  MoveL 5894 to (-63.02, -0.01, -9) mm, rotated rx -180 ry 0 rz 90 deg; joints [73.202, -18.477, 88.716, 0, 19.76, 73.202]
  MoveL 5895 to (-27.01, 8.34, -9) mm, rotated rx -180 ry 0 rz 90 deg; joints [73.832, -17.933, 86.424, 0, 21.509, 73.832]
  MoveL 5896 to (-22.05, 9.5, -9) mm, rotated rx 180 ry 0 rz 90 deg; joints [73.917, -17.854, 86.103, 0, 21.751, 73.917]
  MoveC 5897 to (-21.12, 9.91, -9) mm, rotated rx 180 ry 0 rz 90 deg; joints [73.939, -17.84, 86.046, 0, 21.794, 73.939] to (-20.37, 10.6, -9) mm, rotated rx 180 ry 0 rz 90 deg; joints [73.969, -17.83, 86.008, 0, 21.822, 73.969]
  MoveC 5898 to (-19.58, 12.14, -9) mm, rotated rx -180 ry 0 rz 90 deg; joints [74.027, -17.824, 85.984, 0, 21.841, 74.027] to (-19.7, 13.87, -9) mm, rotated rx 180 ry 0 rz 90 deg; joints [74.082, -17.835, 86.026, 0, 21.809, 74.082]
  MoveL 5899 to (-19.98, 14.69, -9) mm, rotated rx 180 ry 0 rz 90 deg; joints [74.107, -17.844, 86.062, 0, 21.782, 74.107]
  MoveL 5900 to (-26.01, 31.57, -9) mm, rotated rx 180 ry 0 rz 90 deg; joints [74.608, -18.027, 86.81, 0, 21.218, 74.608]
  MoveC 5901 to (-26.34, 32.29, -9) mm, rotated rx 180 ry 0 rz 90 deg; joints [74.628, -18.036, 86.846, 0, 21.19, 74.628] to (-26.8, 32.94, -9) mm, rotated rx -180 ry 0 rz 90 deg; joints [74.646, -18.047, 86.89, 0, 21.156, 74.646]
  MoveL 5902 to (-27.74, 33.64, -9) mm, rotated rx 180 ry 0 rz 90 deg; joints [74.66, -18.066, 86.969, 0, 21.097, 74.66]
  MoveL 5903 to (-62.07, 55.73, -9) mm, rotated rx -180 ry 0 rz 90 deg; joints [75.091, -18.703, 89.719, 0, 18.983, 75.091]
  MoveL 5904 to (-69.19, 60.28, -9) mm, rotated rx 180 ry 0 rz 90 deg; joints [75.181, -18.825, 90.278, 0, 18.547, 75.181]
  MoveC 5905 to (-69.62, 60.48, -9) mm, rotated rx -180 ry 0 rz 90 deg; joints [75.184, -18.832, 90.311, 0, 18.521, 75.184] to (-70.09, 60.56, -9) mm, rotated rx -180 ry 0 rz 90 deg; joints [75.183, -18.84, 90.344, 0, 18.496, 75.183]
  MoveC 5906 to (-72.08, 60.11, -9) mm, rotated rx 180 ry 0 rz 90 deg; joints [75.149, -18.867, 90.469, 0, 18.397, 75.149] to (-73.6, 58.75, -9) mm, rotated rx 180 ry 0 rz 90 deg; joints [75.089, -18.883, 90.547, 0, 18.337, 75.089]
  MoveC 5907 to (-73.89, 58.14, -9) mm, rotated rx 180 ry 0 rz 90 deg; joints [75.065, -18.885, 90.555, 0, 18.33, 75.065] to (-73.99, 57.48, -9) mm, rotated rx -180 ry 0 rz 90 deg; joints [75.042, -18.884, 90.55, 0, 18.334, 75.042]
  MoveL 5908 to (-73.99, 29.63, -9) mm, rotated rx 180 ry 0 rz 90 deg; joints [74.092, -18.773, 90.036, 0, 18.736, 74.092]
  MoveL 5909 to (-66.44, 29.63, -9) mm, rotated rx -180 ry 0 rz 90 deg; joints [74.165, -18.661, 89.531, 0, 19.13, 74.165]
  MoveL 5910 to (-66.44, 29.63, -6) mm, rotated rx -180 ry 0 rz 90 deg; joints [74.165, -18.818, 89.632, 0, 19.185, 74.165]
  Establecer velocidad (1000.0 mm/s)
  MoveL 5911 to (-66.44, 29.63, 10) mm, rotated rx 180 ry 0 rz 90 deg; joints [74.165, -19.655, 90.167, 0, 19.487, 74.165]
  Establecer velocidad (66.7 mm/s)
  MoveL 5912 to (-39.77, -31.53, 10) mm, rotated rx -180 ry 0 rz 90 deg; joints [72.398, -18.924, 87.105, 0, 21.819, 72.398]
  MoveL 5913 to (-39.77, -31.53, -5.75) mm, rotated rx -180 ry 0 rz 90 deg; joints [72.398, -18.112, 86.579, 0, 21.532, 72.398]
  MoveL 5914 to (-39.9, -30.02, -6.16) mm, rotated rx 180 ry 0 rz 90 deg; joints [72.446, -18.101, 86.607, 0, 21.494, 72.446]
  MoveL 5915 to (-40.39, -28.58, -6.56) mm, rotated rx -180 ry 0 rz 90 deg; joints [72.488, -18.096, 86.659, 0, 21.437, 72.488]
  MoveL 5916 to (-41.19, -27.29, -6.97) mm, rotated rx -180 ry 0 rz 90 deg; joints [72.522, -18.095, 86.728, 0, 21.368, 72.522]
  MoveL 5917 to (-42.25, -26.2, -7.38) mm, rotated rx -180 ry 0 rz 90 deg; joints [72.547, -18.098, 86.81, 0, 21.287, 72.547]
  MoveL 5918 to (-43.53, -25.38, -7.78) mm, rotated rx 180 ry 0 rz 90 deg; joints [72.561, -18.102, 86.902, 0, 21.201, 72.561]
  MoveL 5919 to (-44.95, -24.86, -8.19) mm, rotated rx 180 ry 0 rz 90 deg; joints [72.563, -18.108, 86.997, 0, 21.111, 72.563]
  MoveL 5920 to (-46.46, -24.67, -8.59) mm, rotated rx 180 ry 0 rz 90 deg; joints [72.554, -18.113, 87.09, 0, 21.022, 72.554]
  MoveL 5921 to (-47.97, -24.84, -9) mm, rotated rx 180 ry 0 rz 90 deg; joints [72.533, -18.116, 87.176, 0, 20.94, 72.533]
  MoveL 5922 to (-71.48, -29.8, -9) mm, rotated rx -180 ry 0 rz 90 deg; joints [72.121, -18.464, 88.66, 0, 19.804, 72.121]
  MoveC 5923 to (-73.12, -30.73, -9) mm, rotated rx -180 ry 0 rz 90 deg; joints [72.073, -18.485, 88.75, 0, 19.735, 72.073] to (-73.94, -32.43, -9) mm, rotated rx 180 ry 0 rz 90 deg; joints [72.008, -18.489, 88.768, 0, 19.721, 72.008]
  MoveC 5924 to (-73.98, -32.78, -9) mm, rotated rx 180 ry 0 rz 90 deg; joints [71.996, -18.487, 88.763, 0, 19.725, 71.996] to (-73.99, -33.14, -9) mm, rotated rx 180 ry 0 rz 90 deg; joints [71.983, -18.486, 88.756, 0, 19.73, 71.983]
  MoveL 5925 to (-73.99, -70.1, -9) mm, rotated rx 180 ry 0 rz 90 deg; joints [70.765, -18.292, 87.921, 0, 20.371, 70.765]
  MoveC 5926 to (-73.78, -71.26, -9) mm, rotated rx -180 ry 0 rz 90 deg; joints [70.729, -18.283, 87.88, 0, 20.403, 70.729] to (-73.19, -72.29, -9) mm, rotated rx -180 ry 0 rz 90 deg; joints [70.703, -18.268, 87.816, 0, 20.452, 70.703]
  MoveC 5927 to (-72.08, -73.13, -9) mm, rotated rx 180 ry 0 rz 90 deg; joints [70.688, -18.246, 87.722, 0, 20.524, 70.688] to (-70.73, -73.41, -9) mm, rotated rx -180 ry 0 rz 90 deg; joints [70.694, -18.223, 87.624, 0, 20.598, 70.694]
  MoveL 5928 to (-36.48, -73.09, -9) mm, rotated rx 180 ry 0 rz 90 deg; joints [71.089, -17.652, 85.298, 0, 22.355, 71.089]
  MoveL 5929 to (-35.72, -73.07, -9) mm, rotated rx 180 ry 0 rz 90 deg; joints [71.098, -17.639, 85.245, 0, 22.394, 71.098]
  MoveC 5930 to (-33.81, -72.36, -9) mm, rotated rx 180 ry 0 rz 90 deg; joints [71.141, -17.61, 85.13, 0, 22.48, 71.141] to (-32.71, -70.66, -9) mm, rotated rx 180 ry 0 rz 90 deg; joints [71.208, -17.601, 85.094, 0, 22.507, 71.208]
  MoveL 5931 to (-20.54, -23.88, -9) mm, rotated rx 180 ry 0 rz 90 deg; joints [72.843, -17.654, 85.303, 0, 22.351, 72.843]
  MoveC 5932 to (-20.49, -23.55, -9) mm, rotated rx 180 ry 0 rz 90 deg; joints [72.854, -17.655, 85.307, 0, 22.348, 72.854] to (-20.52, -23.22, -9) mm, rotated rx 180 ry 0 rz 90 deg; joints [72.865, -17.657, 85.316, 0, 22.341, 72.865]
  MoveC 5933 to (-21.45, -21.25, -9) mm, rotated rx 180 ry 0 rz 90 deg; joints [72.919, -17.684, 85.423, 0, 22.261, 72.919] to (-23.23, -19.99, -9) mm, rotated rx -180 ry 0 rz 90 deg; joints [72.942, -17.722, 85.574, 0, 22.148, 72.942]
  MoveC 5934 to (-23.83, -19.86, -9) mm, rotated rx 180 ry 0 rz 90 deg; joints [72.941, -17.733, 85.619, 0, 22.114, 72.941] to (-24.45, -19.9, -9) mm, rotated rx 180 ry 0 rz 90 deg; joints [72.933, -17.744, 85.661, 0, 22.083, 72.933]
  MoveL 5935 to (-33.64, -21.82, -9) mm, rotated rx 180 ry 0 rz 90 deg; joints [72.778, -17.892, 86.257, 0, 21.635, 72.778]
  MoveL 5936 to (-47.97, -24.84, -9) mm, rotated rx 180 ry 0 rz 90 deg; joints [72.533, -18.116, 87.176, 0, 20.94, 72.533]
  MoveL 5937 to (-46.41, -32.23, -9) mm, rotated rx 180 ry 0 rz 90 deg; joints [72.307, -18.051, 86.909, 0, 21.142, 72.307]
  MoveL 5938 to (-46.41, -32.23, -6) mm, rotated rx -180 ry 0 rz 90 deg; joints [72.307, -18.206, 87.011, 0, 21.195, 72.307]
  Establecer velocidad (1000.0 mm/s)
  MoveL 5939 to (-46.41, -32.23, 10) mm, rotated rx -180 ry 0 rz 90 deg; joints [72.307, -19.033, 87.545, 0, 21.488, 72.307]
  Establecer velocidad (66.7 mm/s)
  MoveL 5940 to (15.82, -64.4, 10) mm, rotated rx -180 ry 0 rz 90 deg; joints [71.919, -17.693, 82.448, 0, 25.246, 71.919]
  MoveL 5941 to (15.82, -64.4, -5.75) mm, rotated rx 180 ry 0 rz 90 deg; joints [71.919, -16.896, 81.92, 0, 24.977, 71.919]
  MoveL 5942 to (15.68, -65.91, -6.16) mm, rotated rx 180 ry 0 rz 90 deg; joints [71.87, -16.869, 81.881, 0, 24.988, 71.87]
  MoveL 5943 to (15.9, -67.41, -6.56) mm, rotated rx 180 ry 0 rz 90 deg; joints [71.826, -16.834, 81.815, 0, 25.019, 71.826]
  MoveL 5944 to (16.45, -68.83, -6.97) mm, rotated rx 180 ry 0 rz 90 deg; joints [71.787, -16.793, 81.728, 0, 25.065, 71.787]
  MoveL 5945 to (17.29, -70.09, -7.38) mm, rotated rx 180 ry 0 rz 90 deg; joints [71.756, -16.747, 81.623, 0, 25.124, 71.756]
  MoveL 5946 to (18.4, -71.13, -7.78) mm, rotated rx -180 ry 0 rz 90 deg; joints [71.735, -16.698, 81.504, 0, 25.194, 71.735]
  MoveL 5947 to (19.71, -71.9, -8.19) mm, rotated rx -180 ry 0 rz 90 deg; joints [71.724, -16.646, 81.377, 0, 25.269, 71.724]
  MoveL 5948 to (21.16, -72.36, -8.59) mm, rotated rx 180 ry 0 rz 90 deg; joints [71.725, -16.593, 81.247, 0, 25.346, 71.725]
  MoveL 5949 to (22.67, -72.47, -9) mm, rotated rx -180 ry 0 rz 90 deg; joints [71.737, -16.541, 81.121, 0, 25.42, 71.737]
  MoveC 5950 to (33.77, -72.15, -9) mm, rotated rx -180 ry 0 rz 90 deg; joints [71.861, -16.316, 80.318, 0, 25.998, 71.861] to (44.87, -71.79, -9) mm, rotated rx 180 ry 0 rz 90 deg; joints [71.984, -16.085, 79.509, 0, 26.576, 71.984]
  MoveC 5951 to (46.9, -69.65, -9) mm, rotated rx -180 ry 0 rz 90 deg; joints [72.07, -16.056, 79.41, 0, 26.647, 72.07] to (47.66, -66.81, -9) mm, rotated rx 180 ry 0 rz 90 deg; joints [72.165, -16.06, 79.421, 0, 26.639, 72.165]
  MoveL 5952 to (47.63, -65.95, -9) mm, rotated rx -180 ry 0 rz 90 deg; joints [72.192, -16.066, 79.444, 0, 26.622, 72.192]
  MoveC 5953 to (47.48, -65.22, -9) mm, rotated rx -180 ry 0 rz 90 deg; joints [72.213, -16.074, 79.473, 0, 26.602, 72.213] to (47.1, -64.57, -9) mm, rotated rx 180 ry 0 rz 90 deg; joints [72.229, -16.087, 79.516, 0, 26.571, 72.229]
  MoveL 5954 to (45.03, -62.07, -9) mm, rotated rx -180 ry 0 rz 90 deg; joints [72.286, -16.148, 79.729, 0, 26.419, 72.286]
  MoveL 5955 to (29.13, -43.12, -9) mm, rotated rx -180 ry 0 rz 90 deg; joints [72.72, -16.601, 81.336, 0, 25.265, 72.72]
  MoveL 5956 to (25.02, -38.27, -9) mm, rotated rx -180 ry 0 rz 90 deg; joints [72.833, -16.714, 81.744, 0, 24.969, 72.833]
  MoveC 5957 to (24.6, -37.8, -9) mm, rotated rx -180 ry 0 rz 90 deg; joints [72.844, -16.725, 81.785, 0, 24.94, 72.844] to (24.17, -37.36, -9) mm, rotated rx -180 ry 0 rz 90 deg; joints [72.853, -16.736, 81.826, 0, 24.91, 72.853]
  MoveL 5958 to (12.79, -28.13, -9) mm, rotated rx 180 ry 0 rz 90 deg; joints [73.035, -17.014, 82.851, 0, 24.163, 73.035]
  MoveC 5959 to (10.35, -27.65, -9) mm, rotated rx 180 ry 0 rz 90 deg; joints [73.027, -17.064, 83.037, 0, 24.027, 73.027] to (8.05, -28.61, -9) mm, rotated rx -180 ry 0 rz 90 deg; joints [72.974, -17.102, 83.18, 0, 23.922, 72.974]
  MoveC 5960 to (7.53, -29.2, -9) mm, rotated rx -180 ry 0 rz 90 deg; joints [72.95, -17.109, 83.205, 0, 23.904, 72.95] to (7.21, -29.92, -9) mm, rotated rx 180 ry 0 rz 90 deg; joints [72.924, -17.111, 83.212, 0, 23.899, 72.924]
  MoveL 5961 to (-2.19, -64.91, -9) mm, rotated rx 180 ry 0 rz 90 deg; joints [71.717, -17.078, 83.087, 0, 23.99, 71.717]
  MoveL 5962 to (-3.2, -68.7, -9) mm, rotated rx -180 ry 0 rz 90 deg; joints [71.586, -17.073, 83.069, 0, 24.004, 71.586]
  MoveL 5963 to (-3.29, -69.18, -9) mm, rotated rx -180 ry 0 rz 90 deg; joints [71.57, -17.072, 83.064, 0, 24.007, 71.57]
  MoveC 5964 to (-2.2, -71.85, -9) mm, rotated rx 180 ry 0 rz 90 deg; joints [71.497, -17.034, 82.923, 0, 24.11, 71.497] to (0.47, -72.94, -9) mm, rotated rx 180 ry 0 rz 90 deg; joints [71.491, -16.976, 82.707, 0, 24.269, 71.491]
  MoveC 5965 to (11.57, -72.73, -9) mm, rotated rx 180 ry 0 rz 90 deg; joints [71.614, -16.761, 81.917, 0, 24.844, 71.614] to (22.67, -72.47, -9) mm, rotated rx -180 ry 0 rz 90 deg; joints [71.737, -16.541, 81.121, 0, 25.42, 71.737]
  MoveL 5966 to (22.48, -64.92, -9) mm, rotated rx 180 ry 0 rz 90 deg; joints [71.971, -16.595, 81.315, 0, 25.28, 71.971]
  MoveL 5967 to (22.48, -64.92, -6) mm, rotated rx -180 ry 0 rz 90 deg; joints [71.971, -16.747, 81.417, 0, 25.33, 71.971]
  Establecer velocidad (1000.0 mm/s)
  MoveL 5968 to (22.48, -64.92, 10) mm, rotated rx 180 ry 0 rz 90 deg; joints [71.971, -17.555, 81.954, 0, 25.601, 71.971]
  Establecer velocidad (66.7 mm/s)
  MoveL 5969 to (59.51, -30.19, 10) mm, rotated rx 180 ry 0 rz 90 deg; joints [73.413, -17.003, 80.025, 0, 26.978, 73.413]
  MoveL 5970 to (59.51, -30.19, -5.75) mm, rotated rx 180 ry 0 rz 90 deg; joints [73.413, -16.212, 79.495, 0, 26.718, 73.413]
  MoveL 5971 to (60.85, -30.9, -6.16) mm, rotated rx 180 ry 0 rz 90 deg; joints [73.403, -16.158, 79.364, 0, 26.794, 73.403]
  MoveL 5972 to (62.34, -31.19, -6.56) mm, rotated rx 180 ry 0 rz 90 deg; joints [73.408, -16.103, 79.232, 0, 26.871, 73.408]
  MoveL 5973 to (63.86, -31.07, -6.97) mm, rotated rx -180 ry 0 rz 90 deg; joints [73.426, -16.051, 79.107, 0, 26.943, 73.426]
  MoveL 5974 to (65.28, -30.55, -7.38) mm, rotated rx 180 ry 0 rz 90 deg; joints [73.455, -16.003, 78.998, 0, 27.005, 73.455]
  MoveL 5975 to (66.52, -29.67, -7.78) mm, rotated rx 180 ry 0 rz 90 deg; joints [73.494, -15.961, 78.911, 0, 27.05, 73.494]
  MoveL 5976 to (67.47, -28.48, -8.19) mm, rotated rx 180 ry 0 rz 90 deg; joints [73.539, -15.927, 78.851, 0, 27.076, 73.539]
  MoveL 5977 to (68.07, -27.09, -8.59) mm, rotated rx 180 ry 0 rz 90 deg; joints [73.588, -15.903, 78.823, 0, 27.08, 73.588]
  MoveL 5978 to (68.25, -25.58, -9) mm, rotated rx 180 ry 0 rz 90 deg; joints [73.636, -15.888, 78.829, 0, 27.059, 73.636]
  MoveL 5979 to (68.25, -25.3, -9) mm, rotated rx -180 ry 0 rz 90 deg; joints [73.645, -15.89, 78.836, 0, 27.055, 73.645]
  MoveL 5980 to (68.25, -16, -9) mm, rotated rx -180 ry 0 rz 90 deg; joints [73.933, -15.949, 79.039, 0, 26.91, 73.933]
  MoveC 5981 to (66.24, -14.77, -9) mm, rotated rx -180 ry 0 rz 90 deg; joints [73.954, -16.001, 79.217, 0, 26.784, 73.954] to (63.9, -14.53, -9) mm, rotated rx 180 ry 0 rz 90 deg; joints [73.94, -16.053, 79.398, 0, 26.655, 73.94]
  MoveL 5982 to (56.93, -23.93, -9) mm, rotated rx -180 ry 0 rz 90 deg; joints [73.584, -16.144, 79.714, 0, 26.43, 73.584]
  MoveC 5983 to (56.31, -25.98, -9) mm, rotated rx 180 ry 0 rz 90 deg; joints [73.514, -16.144, 79.715, 0, 26.429, 73.514] to (57.13, -27.96, -9) mm, rotated rx -180 ry 0 rz 90 deg; joints [73.46, -16.114, 79.611, 0, 26.504, 73.46]
  MoveL 5984 to (57.98, -28.9, -9) mm, rotated rx -180 ry 0 rz 90 deg; joints [73.439, -16.09, 79.526, 0, 26.564, 73.439]
  MoveL 5985 to (64.27, -35.87, -9) mm, rotated rx 180 ry 0 rz 90 deg; joints [73.281, -15.908, 78.899, 0, 27.01, 73.281]
  MoveC 5986 to (66.4, -35.67, -9) mm, rotated rx 180 ry 0 rz 90 deg; joints [73.307, -15.863, 78.743, 0, 27.12, 73.307] to (68.25, -34.59, -9) mm, rotated rx -180 ry 0 rz 90 deg; joints [73.357, -15.83, 78.628, 0, 27.202, 73.357]
  MoveL 5987 to (68.25, -25.3, -9) mm, rotated rx -180 ry 0 rz 90 deg; joints [73.645, -15.89, 78.836, 0, 27.055, 73.645]
  MoveL 5988 to (60.7, -25.3, -9) mm, rotated rx -180 ry 0 rz 90 deg; joints [73.576, -16.054, 79.403, 0, 26.652, 73.576]
  MoveL 5989 to (60.7, -25.3, -6) mm, rotated rx 180 ry 0 rz 90 deg; joints [73.576, -16.205, 79.505, 0, 26.7, 73.576]
  Establecer velocidad (1000.0 mm/s)
  MoveL 5990 to (60.7, -25.3, 10) mm, rotated rx -180 ry 0 rz 90 deg; joints [73.576, -17.008, 80.044, 0, 26.964, 73.576]
  Establecer velocidad (66.7 mm/s)
  MoveL 5991 to (35.81, 19.66, 10) mm, rotated rx 180 ry 0 rz 90 deg; joints [74.771, -17.797, 82.822, 0, 24.975, 74.771]
  MoveL 5992 to (35.81, 19.66, -5.75) mm, rotated rx 180 ry 0 rz 90 deg; joints [74.771, -16.999, 82.294, 0, 24.705, 74.771]
  MoveL 5993 to (35.98, 21.17, -6.16) mm, rotated rx 180 ry 0 rz 90 deg; joints [74.82, -16.983, 82.297, 0, 24.685, 74.82]
  MoveL 5994 to (35.79, 22.67, -6.56) mm, rotated rx 180 ry 0 rz 90 deg; joints [74.867, -16.974, 82.328, 0, 24.646, 74.867]
  MoveL 5995 to (35.26, 24.1, -6.97) mm, rotated rx -180 ry 0 rz 90 deg; joints [74.908, -16.972, 82.381, 0, 24.591, 74.908]
  MoveL 5996 to (34.43, 25.37, -7.38) mm, rotated rx 180 ry 0 rz 90 deg; joints [74.941, -16.974, 82.452, 0, 24.522, 74.941]
  MoveL 5997 to (33.34, 26.43, -7.78) mm, rotated rx -180 ry 0 rz 90 deg; joints [74.966, -16.981, 82.538, 0, 24.443, 74.966]
  MoveL 5998 to (32.04, 27.22, -8.19) mm, rotated rx -180 ry 0 rz 90 deg; joints [74.98, -16.99, 82.634, 0, 24.356, 74.98]
  MoveL 5999 to (30.6, 27.71, -8.59) mm, rotated rx 180 ry 0 rz 90 deg; joints [74.983, -17, 82.735, 0, 24.265, 74.983]
  MoveL 6000 to (29.09, 27.83, -9) mm, rotated rx 180 ry 0 rz 90 deg; joints [74.974, -17.01, 82.833, 0, 24.177, 74.974]
  MoveC 6001 to (20.47, 27.73, -9) mm, rotated rx -180 ry 0 rz 90 deg; joints [74.896, -17.175, 83.454, 0, 23.721, 74.896] to (11.85, 27.59, -9) mm, rotated rx -180 ry 0 rz 90 deg; joints [74.816, -17.337, 84.069, 0, 23.267, 74.816]
  MoveC 6002 to (9.17, 26.16, -9) mm, rotated rx 180 ry 0 rz 90 deg; joints [74.746, -17.379, 84.233, 0, 23.147, 74.746] to (8.4, 23.22, -9) mm, rotated rx 180 ry 0 rz 90 deg; joints [74.644, -17.379, 84.23, 0, 23.149, 74.644]
  MoveL 6003 to (8.59, 22.68, -9) mm, rotated rx 180 ry 0 rz 90 deg; joints [74.628, -17.372, 84.206, 0, 23.166, 74.628]
  MoveL 6004 to (13.11, 10.33, -9) mm, rotated rx 180 ry 0 rz 90 deg; joints [74.269, -17.224, 83.637, 0, 23.586, 74.269]
  MoveC 6005 to (13.52, 9.55, -9) mm, rotated rx -180 ry 0 rz 90 deg; joints [74.248, -17.212, 83.592, 0, 23.619, 74.248] to (14.12, 8.91, -9) mm, rotated rx 180 ry 0 rz 90 deg; joints [74.233, -17.197, 83.536, 0, 23.661, 74.233]
  MoveL 6006 to (14.69, 8.46, -9) mm, rotated rx 180 ry 0 rz 90 deg; joints [74.224, -17.184, 83.486, 0, 23.697, 74.224]
  MoveL 6007 to (27.9, -1.55, -9) mm, rotated rx 180 ry 0 rz 90 deg; joints [74.024, -16.873, 82.328, 0, 24.545, 74.024]
  MoveC 6008 to (28.39, -1.91, -9) mm, rotated rx 180 ry 0 rz 90 deg; joints [74.017, -16.862, 82.285, 0, 24.577, 74.017] to (28.9, -2.24, -9) mm, rotated rx -180 ry 0 rz 90 deg; joints [74.011, -16.85, 82.241, 0, 24.609, 74.011]
  MoveC 6009 to (31.51, -2.31, -9) mm, rotated rx -180 ry 0 rz 90 deg; joints [74.032, -16.798, 82.05, 0, 24.747, 74.032] to (33.64, -0.82, -9) mm, rotated rx 180 ry 0 rz 90 deg; joints [74.099, -16.763, 81.926, 0, 24.838, 74.099]
  MoveL 6010 to (33.89, -0.47, -9) mm, rotated rx 180 ry 0 rz 90 deg; joints [74.112, -16.761, 81.915, 0, 24.846, 74.112]
  MoveL 6011 to (49.12, 21.32, -9) mm, rotated rx 180 ry 0 rz 90 deg; joints [74.938, -16.574, 81.24, 0, 25.334, 74.938]
  MoveC 6012 to (48.88, 25.12, -9) mm, rotated rx 180 ry 0 rz 90 deg; joints [75.057, -16.6, 81.333, 0, 25.267, 75.057] to (46.33, 27.95, -9) mm, rotated rx -180 ry 0 rz 90 deg; joints [75.125, -16.667, 81.576, 0, 25.092, 75.125]
  MoveC 6013 to (37.71, 27.91, -9) mm, rotated rx -180 ry 0 rz 90 deg; joints [75.05, -16.84, 82.207, 0, 24.633, 75.05] to (29.09, 27.83, -9) mm, rotated rx 180 ry 0 rz 90 deg; joints [74.974, -17.01, 82.833, 0, 24.177, 74.974]
  MoveL 6014 to (29.17, 20.28, -9) mm, rotated rx 180 ry 0 rz 90 deg; joints [74.732, -16.968, 82.679, 0, 24.289, 74.732]
  MoveL 6015 to (29.17, 20.28, -6) mm, rotated rx 180 ry 0 rz 90 deg; joints [74.732, -17.121, 82.781, 0, 24.34, 74.732]
  Establecer velocidad (1000.0 mm/s)
  MoveL 6016 to (29.17, 20.28, 10) mm, rotated rx 180 ry 0 rz 90 deg; joints [74.732, -17.933, 83.317, 0, 24.616, 74.732]
  Establecer velocidad (66.7 mm/s)
  MoveL 6017 to (29.13, 63.8, 10) mm, rotated rx -180 ry 0 rz 90 deg; joints [76.136, -18.156, 84.138, 0, 24.017, 76.136]
  MoveL 6018 to (29.13, 63.8, -5.75) mm, rotated rx 180 ry 0 rz 90 deg; joints [76.136, -17.353, 83.611, 0, 23.742, 76.136]
  MoveL 6019 to (29.35, 65.3, -6.16) mm, rotated rx -180 ry 0 rz 90 deg; joints [76.186, -17.335, 83.608, 0, 23.727, 76.186]
  MoveL 6020 to (29.21, 66.81, -6.56) mm, rotated rx 180 ry 0 rz 90 deg; joints [76.234, -17.324, 83.632, 0, 23.693, 76.234]
  MoveL 6021 to (28.74, 68.26, -6.97) mm, rotated rx -180 ry 0 rz 90 deg; joints [76.278, -17.32, 83.678, 0, 23.642, 76.278]
  MoveL 6022 to (27.96, 69.56, -7.38) mm, rotated rx -180 ry 0 rz 90 deg; joints [76.314, -17.32, 83.743, 0, 23.577, 76.314]
  MoveL 6023 to (26.9, 70.66, -7.78) mm, rotated rx -180 ry 0 rz 90 deg; joints [76.341, -17.324, 83.825, 0, 23.5, 76.341]
  MoveL 6024 to (25.63, 71.49, -8.19) mm, rotated rx -180 ry 0 rz 90 deg; joints [76.358, -17.331, 83.917, 0, 23.414, 76.358]
  MoveL 6025 to (24.21, 72.03, -8.59) mm, rotated rx -180 ry 0 rz 90 deg; joints [76.365, -17.34, 84.015, 0, 23.325, 76.365]
  MoveL 6026 to (22.71, 72.21, -9) mm, rotated rx 180 ry 0 rz 90 deg; joints [76.359, -17.348, 84.113, 0, 23.235, 76.359]
  MoveC 6027 to (0.28, 72.74, -9) mm, rotated rx 180 ry 0 rz 90 deg; joints [76.196, -17.759, 85.72, 0, 22.039, 76.196] to (-22.14, 73.15, -9) mm, rotated rx -180 ry 0 rz 90 deg; joints [76.025, -18.145, 87.297, 0, 20.848, 76.025]
  MoveC 6028 to (-24.58, 70.15, -9) mm, rotated rx 180 ry 0 rz 90 deg; joints [75.905, -18.172, 87.414, 0, 20.759, 75.905] to (-24.23, 66.3, -9) mm, rotated rx 180 ry 0 rz 90 deg; joints [75.779, -18.151, 87.323, 0, 20.828, 75.779]
  MoveL 6029 to (-8.76, 56.39, -9) mm, rotated rx 180 ry 0 rz 90 deg; joints [75.58, -17.845, 86.067, 0, 21.778, 75.58]
  MoveL 6030 to (-7.82, 55.83, -9) mm, rotated rx -180 ry 0 rz 90 deg; joints [75.57, -17.826, 85.991, 0, 21.835, 75.57]
  MoveC 6031 to (-7.56, 55.72, -9) mm, rotated rx 180 ry 0 rz 90 deg; joints [75.569, -17.821, 85.971, 0, 21.85, 75.569] to (-7.28, 55.7, -9) mm, rotated rx 180 ry 0 rz 90 deg; joints [75.57, -17.816, 85.951, 0, 21.865, 75.57]
  MoveC 6032 to (-2.66, 56.02, -9) mm, rotated rx 180 ry 0 rz 90 deg; joints [75.62, -17.736, 85.631, 0, 22.105, 75.62] to (1.96, 56.39, -9) mm, rotated rx -180 ry 0 rz 90 deg; joints [75.671, -17.656, 85.312, 0, 22.344, 75.671]
  MoveC 6033 to (20.66, 57.9, -9) mm, rotated rx 180 ry 0 rz 90 deg; joints [75.876, -17.32, 84.006, 0, 23.315, 75.876] to (39.33, 59.8, -9) mm, rotated rx 180 ry 0 rz 90 deg; joints [76.088, -16.971, 82.688, 0, 24.282, 76.088]
  MoveC 6034 to (53.26, 61.6, -9) mm, rotated rx -180 ry 0 rz 90 deg; joints [76.256, -16.701, 81.698, 0, 25.003, 76.256] to (67.12, 63.92, -9) mm, rotated rx -180 ry 0 rz 90 deg; joints [76.438, -16.426, 80.71, 0, 25.716, 76.438]
  MoveC 6035 to (67.71, 64.09, -9) mm, rotated rx -180 ry 0 rz 90 deg; joints [76.448, -16.415, 80.669, 0, 25.746, 76.448] to (68.25, 64.38, -9) mm, rotated rx -180 ry 0 rz 90 deg; joints [76.461, -16.405, 80.634, 0, 25.771, 76.461]
  MoveL 6036 to (68.25, 69.29, -9) mm, rotated rx 180 ry 0 rz 90 deg; joints [76.617, -16.43, 80.722, 0, 25.708, 76.617]
  MoveC 6037 to (67.9, 69.52, -9) mm, rotated rx 180 ry 0 rz 90 deg; joints [76.622, -16.438, 80.753, 0, 25.686, 76.622] to (67.48, 69.63, -9) mm, rotated rx 180 ry 0 rz 90 deg; joints [76.622, -16.447, 80.785, 0, 25.662, 76.622]
  MoveC 6038 to (45.37, 71.28, -9) mm, rotated rx -180 ry 0 rz 90 deg; joints [76.506, -16.907, 82.451, 0, 24.456, 76.506] to (23.22, 72.19, -9) mm, rotated rx -180 ry 0 rz 90 deg; joints [76.362, -17.338, 84.076, 0, 23.263, 76.362]
  MoveC 6039 to (22.96, 72.2, -9) mm, rotated rx -180 ry 0 rz 90 deg; joints [76.36, -17.343, 84.094, 0, 23.249, 76.36] to (22.71, 72.21, -9) mm, rotated rx 180 ry 0 rz 90 deg; joints [76.359, -17.348, 84.113, 0, 23.235, 76.359]
  MoveL 6040 to (22.51, 64.66, -9) mm, rotated rx 180 ry 0 rz 90 deg; joints [76.111, -17.317, 83.994, 0, 23.323, 76.111]
  MoveL 6041 to (13.82, 64.88, -9) mm, rotated rx 180 ry 0 rz 90 deg; joints [76.047, -17.48, 84.621, 0, 22.859, 76.047]
  MoveL 6042 to (13.82, 64.88, -6) mm, rotated rx -180 ry 0 rz 90 deg; joints [76.047, -17.633, 84.723, 0, 22.911, 76.047]
  Establecer velocidad (1000.0 mm/s)
  MoveL 6043 to (13.82, 64.88, 10) mm, rotated rx 180 ry 0 rz 90 deg; joints [76.047, -18.452, 85.257, 0, 23.195, 76.047]
  Establecer velocidad (66.7 mm/s)
  MoveL 6044 to (29.12, 63.57, 10) mm, rotated rx -180 ry 0 rz 90 deg; joints [76.128, -18.155, 84.135, 0, 24.02, 76.128]
  MoveL 6045 to (29.12, 63.57, -6) mm, rotated rx 180 ry 0 rz 90 deg; joints [76.128, -17.34, 83.6, 0, 23.74, 76.128]
  MoveL 6046 to (29.34, 65.07, -6.41) mm, rotated rx -180 ry 0 rz 90 deg; joints [76.179, -17.322, 83.596, 0, 23.725, 76.179]
  MoveL 6047 to (29.2, 66.58, -6.81) mm, rotated rx -180 ry 0 rz 90 deg; joints [76.227, -17.311, 83.62, 0, 23.691, 76.227]
  MoveL 6048 to (28.73, 68.03, -7.22) mm, rotated rx -180 ry 0 rz 90 deg; joints [76.27, -17.306, 83.666, 0, 23.64, 76.27]
  MoveL 6049 to (27.95, 69.33, -7.63) mm, rotated rx 180 ry 0 rz 90 deg; joints [76.306, -17.306, 83.731, 0, 23.575, 76.306]
  MoveL 6050 to (26.9, 70.43, -8.03) mm, rotated rx -180 ry 0 rz 90 deg; joints [76.334, -17.31, 83.813, 0, 23.498, 76.334]
  MoveL 6051 to (25.63, 71.27, -8.44) mm, rotated rx 180 ry 0 rz 90 deg; joints [76.351, -17.318, 83.905, 0, 23.413, 76.351]
  MoveL 6052 to (24.21, 71.81, -8.84) mm, rotated rx -180 ry 0 rz 90 deg; joints [76.357, -17.326, 84.003, 0, 23.323, 76.357]
  MoveL 6053 to (22.7, 71.99, -9.25) mm, rotated rx 180 ry 0 rz 90 deg; joints [76.351, -17.334, 84.101, 0, 23.234, 76.351]
  MoveC 6054 to (21.54, 72.02, -9.25) mm, rotated rx -180 ry 0 rz 90 deg; joints [76.343, -17.356, 84.185, 0, 23.171, 76.343] to (20.37, 72.04, -9.25) mm, rotated rx 180 ry 0 rz 90 deg; joints [76.335, -17.378, 84.269, 0, 23.109, 76.335]
  MoveC 6055 to (-0.57, 72.54, -9.25) mm, rotated rx -180 ry 0 rz 90 deg; joints [76.183, -17.76, 85.768, 0, 21.991, 76.183] to (-21.52, 72.95, -9.25) mm, rotated rx -180 ry 0 rz 90 deg; joints [76.024, -18.12, 87.241, 0, 20.879, 76.024]
  MoveC 6056 to (-23.93, 69.99, -9.25) mm, rotated rx -180 ry 0 rz 90 deg; joints [75.904, -18.148, 87.358, 0, 20.79, 75.904] to (-23.6, 66.17, -9.25) mm, rotated rx -180 ry 0 rz 90 deg; joints [75.78, -18.127, 87.268, 0, 20.859, 75.78]
  MoveL 6057 to (-7.79, 56.05, -9.25) mm, rotated rx 180 ry 0 rz 90 deg; joints [75.577, -17.814, 85.984, 0, 21.829, 75.577]
  MoveC 6058 to (-7.44, 55.89, -9.25) mm, rotated rx 180 ry 0 rz 90 deg; joints [75.575, -17.807, 85.957, 0, 21.85, 75.575] to (-7.05, 55.85, -9.25) mm, rotated rx -180 ry 0 rz 90 deg; joints [75.577, -17.8, 85.929, 0, 21.871, 75.577]
  MoveL 6059 to (-5.21, 55.96, -9.25) mm, rotated rx -180 ry 0 rz 90 deg; joints [75.596, -17.768, 85.802, 0, 21.966, 75.596]
  MoveL 6060 to (6.16, 56.85, -9.25) mm, rotated rx -180 ry 0 rz 90 deg; joints [75.721, -17.57, 85.014, 0, 22.556, 75.721]
  MoveC 6061 to (23.71, 58.37, -9.25) mm, rotated rx 180 ry 0 rz 90 deg; joints [75.916, -17.252, 83.786, 0, 23.466, 75.916] to (41.22, 60.26, -9.25) mm, rotated rx 180 ry 0 rz 90 deg; joints [76.118, -16.923, 82.55, 0, 24.373, 76.118]
  MoveC 6062 to (53.34, 61.9, -9.25) mm, rotated rx -180 ry 0 rz 90 deg; joints [76.266, -16.688, 81.689, 0, 24.999, 76.266] to (65.39, 63.96, -9.25) mm, rotated rx -180 ry 0 rz 90 deg; joints [76.426, -16.45, 80.831, 0, 25.619, 76.426]
  MoveL 6063 to (65.39, 69.5, -9.25) mm, rotated rx 180 ry 0 rz 90 deg; joints [76.602, -16.478, 80.931, 0, 25.547, 76.602]
  MoveC 6064 to (44.07, 71.08, -9.25) mm, rotated rx 180 ry 0 rz 90 deg; joints [76.489, -16.919, 82.534, 0, 24.384, 76.489] to (22.7, 71.99, -9.25) mm, rotated rx 180 ry 0 rz 90 deg; joints [76.351, -17.334, 84.101, 0, 23.234, 76.351]
  MoveL 6065 to (22.5, 64.44, -9.25) mm, rotated rx -180 ry 0 rz 90 deg; joints [76.103, -17.303, 83.982, 0, 23.321, 76.103]
  MoveL 6066 to (10.29, 64.74, -9.25) mm, rotated rx -180 ry 0 rz 90 deg; joints [76.014, -17.531, 84.862, 0, 22.669, 76.014]
  MoveL 6067 to (10.29, 64.74, -6.25) mm, rotated rx 180 ry 0 rz 90 deg; joints [76.014, -17.685, 84.964, 0, 22.721, 76.014]
  Establecer velocidad (1000.0 mm/s)
  MoveL 6068 to (10.29, 64.74, 10) mm, rotated rx 180 ry 0 rz 90 deg; joints [76.014, -18.517, 85.507, 0, 23.01, 76.014]
  Establecer velocidad (66.7 mm/s)
  MoveL 6069 to (35.58, 19.41, 10) mm, rotated rx 180 ry 0 rz 90 deg; joints [74.76, -17.8, 82.834, 0, 24.967, 74.76]
  MoveL 6070 to (35.58, 19.41, -6) mm, rotated rx -180 ry 0 rz 90 deg; joints [74.76, -16.989, 82.297, 0, 24.692, 74.76]
  MoveL 6071 to (35.75, 20.92, -6.41) mm, rotated rx -180 ry 0 rz 90 deg; joints [74.81, -16.974, 82.301, 0, 24.672, 74.81]
  MoveL 6072 to (35.55, 22.42, -6.81) mm, rotated rx 180 ry 0 rz 90 deg; joints [74.857, -16.965, 82.331, 0, 24.634, 74.857]
  MoveL 6073 to (35.03, 23.85, -7.22) mm, rotated rx -180 ry 0 rz 90 deg; joints [74.898, -16.962, 82.384, 0, 24.578, 74.898]
  MoveL 6074 to (34.2, 25.12, -7.63) mm, rotated rx -180 ry 0 rz 90 deg; joints [74.931, -16.965, 82.455, 0, 24.509, 74.931]
  MoveL 6075 to (33.11, 26.18, -8.03) mm, rotated rx -180 ry 0 rz 90 deg; joints [74.956, -16.971, 82.542, 0, 24.43, 74.956]
  MoveL 6076 to (31.81, 26.97, -8.44) mm, rotated rx 180 ry 0 rz 90 deg; joints [74.97, -16.98, 82.638, 0, 24.343, 74.97]
  MoveL 6077 to (30.37, 27.46, -8.84) mm, rotated rx -180 ry 0 rz 90 deg; joints [74.973, -16.99, 82.738, 0, 24.253, 74.973]
  MoveL 6078 to (28.86, 27.59, -9.25) mm, rotated rx -180 ry 0 rz 90 deg; joints [74.964, -17, 82.836, 0, 24.164, 74.964]
  MoveC 6079 to (20.35, 27.49, -9.25) mm, rotated rx 180 ry 0 rz 90 deg; joints [74.887, -17.163, 83.449, 0, 23.715, 74.887] to (11.85, 27.35, -9.25) mm, rotated rx 180 ry 0 rz 90 deg; joints [74.808, -17.323, 84.056, 0, 23.267, 74.808]
  MoveC 6080 to (9.44, 25.92, -9.25) mm, rotated rx -180 ry 0 rz 90 deg; joints [74.741, -17.36, 84.2, 0, 23.16, 74.741] to (8.68, 23.22, -9.25) mm, rotated rx -180 ry 0 rz 90 deg; joints [74.646, -17.361, 84.202, 0, 23.159, 74.646]
  MoveL 6081 to (8.82, 22.74, -9.25) mm, rotated rx 180 ry 0 rz 90 deg; joints [74.632, -17.356, 84.182, 0, 23.173, 74.632]
  MoveL 6082 to (12.8, 11.85, -9.25) mm, rotated rx 180 ry 0 rz 90 deg; joints [74.316, -17.225, 83.681, 0, 23.543, 74.316]
  MoveL 6083 to (13.33, 10.44, -9.25) mm, rotated rx -180 ry 0 rz 90 deg; joints [74.275, -17.207, 83.615, 0, 23.592, 74.275]
  MoveC 6084 to (13.74, 9.67, -9.25) mm, rotated rx -180 ry 0 rz 90 deg; joints [74.254, -17.195, 83.571, 0, 23.625, 74.254] to (14.34, 9.03, -9.25) mm, rotated rx 180 ry 0 rz 90 deg; joints [74.239, -17.181, 83.515, 0, 23.666, 74.239]
  MoveL 6085 to (14.69, 8.75, -9.25) mm, rotated rx 180 ry 0 rz 90 deg; joints [74.233, -17.172, 83.484, 0, 23.689, 74.233]
  MoveL 6086 to (28.4, -1.62, -9.25) mm, rotated rx 180 ry 0 rz 90 deg; joints [74.026, -16.85, 82.281, 0, 24.569, 74.026]
  MoveC 6087 to (29.07, -1.99, -9.25) mm, rotated rx 180 ry 0 rz 90 deg; joints [74.02, -16.835, 82.225, 0, 24.61, 74.02] to (29.82, -2.16, -9.25) mm, rotated rx 180 ry 0 rz 90 deg; joints [74.021, -16.819, 82.167, 0, 24.652, 74.021]
  MoveC 6088 to (31.96, -1.8, -9.25) mm, rotated rx 180 ry 0 rz 90 deg; joints [74.053, -16.779, 82.019, 0, 24.76, 74.053] to (33.64, -0.41, -9.25) mm, rotated rx 180 ry 0 rz 90 deg; joints [74.112, -16.753, 81.925, 0, 24.828, 74.112]
  MoveL 6089 to (47.86, 19.95, -9.25) mm, rotated rx 180 ry 0 rz 90 deg; joints [74.884, -16.58, 81.297, 0, 25.283, 74.884]
  MoveL 6090 to (48.38, 20.73, -9.25) mm, rotated rx 180 ry 0 rz 90 deg; joints [74.913, -16.573, 81.274, 0, 25.3, 74.913]
  MoveC 6091 to (48.85, 21.82, -9.25) mm, rotated rx -180 ry 0 rz 90 deg; joints [74.952, -16.57, 81.261, 0, 25.309, 74.952] to (48.86, 23.01, -9.25) mm, rotated rx 180 ry 0 rz 90 deg; joints [74.989, -16.576, 81.284, 0, 25.292, 74.989]
  MoveL 6092 to (48.7, 23.86, -9.25) mm, rotated rx 180 ry 0 rz 90 deg; joints [75.015, -16.584, 81.313, 0, 25.271, 75.015]
  MoveC 6093 to (47.72, 26.09, -9.25) mm, rotated rx 180 ry 0 rz 90 deg; joints [75.077, -16.616, 81.429, 0, 25.188, 75.077] to (45.88, 27.68, -9.25) mm, rotated rx -180 ry 0 rz 90 deg; joints [75.113, -16.662, 81.595, 0, 25.067, 75.113]
  MoveC 6094 to (37.37, 27.65, -9.25) mm, rotated rx 180 ry 0 rz 90 deg; joints [75.039, -16.833, 82.218, 0, 24.615, 75.039] to (28.86, 27.59, -9.25) mm, rotated rx -180 ry 0 rz 90 deg; joints [74.964, -17, 82.836, 0, 24.164, 74.964]
  MoveL 6095 to (28.94, 20.04, -9.25) mm, rotated rx 180 ry 0 rz 90 deg; joints [74.722, -16.959, 82.682, 0, 24.276, 74.722]
  MoveL 6096 to (28.94, 20.04, -6.25) mm, rotated rx 180 ry 0 rz 90 deg; joints [74.722, -17.111, 82.785, 0, 24.327, 74.722]
  Establecer velocidad (1000.0 mm/s)
  MoveL 6097 to (28.94, 20.04, 10) mm, rotated rx 180 ry 0 rz 90 deg; joints [74.722, -17.936, 83.329, 0, 24.608, 74.722]
  Establecer velocidad (66.7 mm/s)
  MoveL 6098 to (63.52, -34.61, 10) mm, rotated rx -180 ry 0 rz 90 deg; joints [73.313, -16.886, 79.626, 0, 27.26, 73.313]
  MoveL 6099 to (63.52, -34.61, -6) mm, rotated rx -180 ry 0 rz 90 deg; joints [73.313, -16.084, 79.086, 0, 26.997, 73.313]
  MoveL 6100 to (64.11, -35.27, -6.24) mm, rotated rx -180 ry 0 rz 90 deg; joints [73.298, -16.055, 79.019, 0, 27.036, 73.298]
  MoveL 6101 to (65.39, -35.25, -6.58) mm, rotated rx 180 ry 0 rz 90 deg; joints [73.311, -16.01, 78.912, 0, 27.098, 73.311]
  MoveL 6102 to (65.39, -25.28, -9.25) mm, rotated rx 180 ry 0 rz 90 deg; joints [73.62, -15.94, 79.042, 0, 26.898, 73.62]
  MoveL 6103 to (65.39, -15.31, -9.25) mm, rotated rx 180 ry 0 rz 90 deg; joints [73.929, -16.003, 79.26, 0, 26.743, 73.929]
  MoveL 6104 to (63.72, -15.23, -9.25) mm, rotated rx 180 ry 0 rz 90 deg; joints [73.917, -16.04, 79.388, 0, 26.652, 73.917]
  MoveL 6105 to (57.33, -23.83, -9.25) mm, rotated rx 180 ry 0 rz 90 deg; joints [73.591, -16.123, 79.678, 0, 26.445, 73.591]
  MoveC 6106 to (56.63, -25.92, -9.25) mm, rotated rx -180 ry 0 rz 90 deg; joints [73.519, -16.125, 79.684, 0, 26.441, 73.519] to (57.48, -27.96, -9.25) mm, rotated rx 180 ry 0 rz 90 deg; joints [73.464, -16.094, 79.576, 0, 26.518, 73.464]
  MoveL 6107 to (64.11, -35.27, -9.25) mm, rotated rx -180 ry 0 rz 90 deg; joints [73.298, -15.903, 78.915, 0, 26.988, 73.298]
  MoveL 6108 to (65.39, -35.25, -9.25) mm, rotated rx -180 ry 0 rz 90 deg; joints [73.311, -15.875, 78.82, 0, 27.055, 73.311]
  MoveL 6109 to (65.39, -25.28, -9.25) mm, rotated rx 180 ry 0 rz 90 deg; joints [73.62, -15.94, 79.042, 0, 26.898, 73.62]
  MoveL 6110 to (57.84, -25.28, -9.25) mm, rotated rx 180 ry 0 rz 90 deg; joints [73.55, -16.103, 79.608, 0, 26.495, 73.55]
  MoveL 6111 to (57.84, -25.28, -6.25) mm, rotated rx 180 ry 0 rz 90 deg; joints [73.55, -16.254, 79.711, 0, 26.544, 73.55]
  Establecer velocidad (1000.0 mm/s)
  MoveL 6112 to (57.84, -25.28, 10) mm, rotated rx 180 ry 0 rz 90 deg; joints [73.55, -17.071, 80.258, 0, 26.812, 73.55]
  Establecer velocidad (66.7 mm/s)
  MoveL 6113 to (15.68, -64.19, 10) mm, rotated rx 180 ry 0 rz 90 deg; joints [71.925, -17.698, 82.462, 0, 25.235, 71.925]
  MoveL 6114 to (15.68, -64.19, -6) mm, rotated rx -180 ry 0 rz 90 deg; joints [71.925, -16.888, 81.926, 0, 24.962, 71.925]
  MoveL 6115 to (15.54, -65.7, -6.41) mm, rotated rx 180 ry 0 rz 90 deg; joints [71.876, -16.86, 81.887, 0, 24.973, 71.876]
  MoveL 6116 to (15.77, -67.2, -6.81) mm, rotated rx -180 ry 0 rz 90 deg; joints [71.831, -16.825, 81.821, 0, 25.004, 71.831]
  MoveL 6117 to (16.32, -68.62, -7.22) mm, rotated rx 180 ry 0 rz 90 deg; joints [71.792, -16.784, 81.734, 0, 25.05, 71.792]
  MoveL 6118 to (17.17, -69.88, -7.63) mm, rotated rx -180 ry 0 rz 90 deg; joints [71.761, -16.739, 81.629, 0, 25.11, 71.761]
  MoveL 6119 to (18.28, -70.92, -8.03) mm, rotated rx 180 ry 0 rz 90 deg; joints [71.74, -16.689, 81.51, 0, 25.179, 71.74]
  MoveL 6120 to (19.59, -71.69, -8.44) mm, rotated rx 180 ry 0 rz 90 deg; joints [71.73, -16.637, 81.383, 0, 25.254, 71.73]
  MoveL 6121 to (21.03, -72.15, -8.84) mm, rotated rx 180 ry 0 rz 90 deg; joints [71.73, -16.584, 81.253, 0, 25.331, 71.73]
  MoveL 6122 to (22.55, -72.24, -9.25) mm, rotated rx -180 ry 0 rz 90 deg; joints [71.743, -16.533, 81.127, 0, 25.406, 71.743]
  MoveC 6123 to (33.47, -71.92, -9.25) mm, rotated rx -180 ry 0 rz 90 deg; joints [71.865, -16.311, 80.338, 0, 25.973, 71.865] to (44.38, -71.53, -9.25) mm, rotated rx -180 ry 0 rz 90 deg; joints [71.987, -16.084, 79.542, 0, 26.542, 71.987]
  MoveC 6124 to (46.76, -68.57, -9.25) mm, rotated rx 180 ry 0 rz 90 deg; joints [72.102, -16.054, 79.437, 0, 26.617, 72.102] to (46.9, -64.78, -9.25) mm, rotated rx 180 ry 0 rz 90 deg; joints [72.221, -16.077, 79.517, 0, 26.56, 72.221]
  MoveC 6125 to (35.85, -51.47, -9.25) mm, rotated rx -180 ry 0 rz 90 deg; joints [72.525, -16.398, 80.645, 0, 25.753, 72.525] to (24.7, -38.23, -9.25) mm, rotated rx -180 ry 0 rz 90 deg; joints [72.831, -16.707, 81.759, 0, 24.948, 72.831]
  MoveC 6126 to (24.23, -37.72, -9.25) mm, rotated rx -180 ry 0 rz 90 deg; joints [72.842, -16.72, 81.805, 0, 24.915, 72.842] to (23.71, -37.26, -9.25) mm, rotated rx 180 ry 0 rz 90 deg; joints [72.852, -16.733, 81.853, 0, 24.88, 72.852]
  MoveL 6127 to (13.54, -29.01, -9.25) mm, rotated rx 180 ry 0 rz 90 deg; joints [73.014, -16.982, 82.77, 0, 24.212, 73.014]
  MoveL 6128 to (13.42, -28.9, -9.25) mm, rotated rx -180 ry 0 rz 90 deg; joints [73.017, -16.985, 82.781, 0, 24.204, 73.017]
  MoveC 6129 to (10.24, -27.99, -9.25) mm, rotated rx -180 ry 0 rz 90 deg; joints [73.015, -17.052, 83.029, 0, 24.023, 73.015] to (7.5, -29.85, -9.25) mm, rotated rx -180 ry 0 rz 90 deg; joints [72.929, -17.093, 83.184, 0, 23.909, 72.929]
  MoveL 6130 to (7.22, -30.8, -9.25) mm, rotated rx 180 ry 0 rz 90 deg; joints [72.896, -17.093, 83.184, 0, 23.909, 72.896]
  MoveL 6131 to (-2.73, -67.76, -9.25) mm, rotated rx 180 ry 0 rz 90 deg; joints [71.621, -17.057, 83.049, 0, 24.008, 71.621]
  MoveL 6132 to (-2.95, -68.7, -9.25) mm, rotated rx 180 ry 0 rz 90 deg; joints [71.589, -17.055, 83.043, 0, 24.012, 71.589]
  MoveC 6133 to (-2.03, -71.54, -9.25) mm, rotated rx 180 ry 0 rz 90 deg; joints [71.509, -17.02, 82.91, 0, 24.109, 71.509] to (0.71, -72.73, -9.25) mm, rotated rx -180 ry 0 rz 90 deg; joints [71.5, -16.96, 82.687, 0, 24.273, 71.5]
  MoveC 6134 to (11.63, -72.51, -9.25) mm, rotated rx 180 ry 0 rz 90 deg; joints [71.622, -16.749, 81.91, 0, 24.839, 71.622] to (22.55, -72.24, -9.25) mm, rotated rx -180 ry 0 rz 90 deg; joints [71.743, -16.533, 81.127, 0, 25.406, 71.743]
  MoveL 6135 to (22.34, -64.7, -9.25) mm, rotated rx 180 ry 0 rz 90 deg; joints [71.977, -16.587, 81.321, 0, 25.265, 71.977]
  MoveL 6136 to (22.34, -64.7, -6.25) mm, rotated rx -180 ry 0 rz 90 deg; joints [71.977, -16.738, 81.424, 0, 25.315, 71.977]
  Establecer velocidad (1000.0 mm/s)
  MoveL 6137 to (22.34, -64.7, 10) mm, rotated rx 180 ry 0 rz 90 deg; joints [71.977, -17.56, 81.969, 0, 25.59, 71.977]
  Establecer velocidad (66.7 mm/s)
  MoveL 6138 to (-36.44, -51.68, 10) mm, rotated rx -180 ry 0 rz 90 deg; joints [71.779, -18.753, 86.427, 0, 22.326, 71.779]
  MoveL 6139 to (-36.44, -51.68, -6) mm, rotated rx -180 ry 0 rz 90 deg; joints [71.779, -17.931, 85.893, 0, 22.038, 71.779]
  MoveL 6140 to (-35.03, -52.23, -6.41) mm, rotated rx 180 ry 0 rz 90 deg; joints [71.776, -17.882, 85.769, 0, 22.113, 71.776]
  MoveL 6141 to (-33.52, -52.44, -6.81) mm, rotated rx 180 ry 0 rz 90 deg; joints [71.785, -17.834, 85.646, 0, 22.188, 71.785]
  MoveL 6142 to (-32.01, -52.3, -7.22) mm, rotated rx 180 ry 0 rz 90 deg; joints [71.806, -17.788, 85.531, 0, 22.256, 71.806]
  MoveL 6143 to (-30.56, -51.83, -7.63) mm, rotated rx -180 ry 0 rz 90 deg; joints [71.836, -17.744, 85.428, 0, 22.316, 71.836]
  MoveL 6144 to (-29.26, -51.06, -8.03) mm, rotated rx 180 ry 0 rz 90 deg; joints [71.875, -17.705, 85.341, 0, 22.364, 71.875]
  MoveL 6145 to (-28.15, -50.01, -8.44) mm, rotated rx 180 ry 0 rz 90 deg; joints [71.92, -17.67, 85.274, 0, 22.396, 71.92]
  MoveL 6146 to (-27.31, -48.75, -8.84) mm, rotated rx 180 ry 0 rz 90 deg; joints [71.97, -17.642, 85.23, 0, 22.412, 71.97]
  MoveL 6147 to (-26.79, -47.32, -9.25) mm, rotated rx 180 ry 0 rz 90 deg; joints [72.021, -17.62, 85.213, 0, 22.407, 72.021]
  MoveL 6148 to (-20.77, -24.15, -9.25) mm, rotated rx -180 ry 0 rz 90 deg; joints [72.832, -17.643, 85.305, 0, 22.339, 72.832]
  MoveC 6149 to (-20.71, -23.68, -9.25) mm, rotated rx -180 ry 0 rz 90 deg; joints [72.848, -17.645, 85.31, 0, 22.334, 72.848] to (-20.77, -23.2, -9.25) mm, rotated rx 180 ry 0 rz 90 deg; joints [72.863, -17.648, 85.325, 0, 22.324, 72.863]
  MoveC 6150 to (-21.66, -21.46, -9.25) mm, rotated rx 180 ry 0 rz 90 deg; joints [72.91, -17.674, 85.424, 0, 22.249, 72.91] to (-23.22, -20.28, -9.25) mm, rotated rx -180 ry 0 rz 90 deg; joints [72.933, -17.707, 85.558, 0, 22.149, 72.933]
  MoveC 6151 to (-23.94, -20.09, -9.25) mm, rotated rx 180 ry 0 rz 90 deg; joints [72.932, -17.721, 85.613, 0, 22.108, 72.932] to (-24.68, -20.12, -9.25) mm, rotated rx 180 ry 0 rz 90 deg; joints [72.924, -17.734, 85.664, 0, 22.07, 72.924]
  MoveL 6152 to (-33.64, -21.99, -9.25) mm, rotated rx -180 ry 0 rz 90 deg; joints [72.773, -17.878, 86.245, 0, 21.633, 72.773]
  MoveL 6153 to (-71.34, -29.93, -9.25) mm, rotated rx -180 ry 0 rz 90 deg; joints [72.119, -18.448, 88.64, 0, 19.809, 72.119]
  MoveC 6154 to (-73.08, -30.98, -9.25) mm, rotated rx -180 ry 0 rz 90 deg; joints [72.065, -18.47, 88.734, 0, 19.736, 72.065] to (-73.8, -32.88, -9.25) mm, rotated rx -180 ry 0 rz 90 deg; joints [71.994, -18.471, 88.74, 0, 19.731, 71.994]
  MoveL 6155 to (-73.83, -33.64, -9.25) mm, rotated rx -180 ry 0 rz 90 deg; joints [71.969, -18.468, 88.725, 0, 19.743, 71.969]
  MoveL 6156 to (-73.83, -70.05, -9.25) mm, rotated rx 180 ry 0 rz 90 deg; joints [70.769, -18.277, 87.903, 0, 20.374, 70.769]
  MoveC 6157 to (-73.34, -71.76, -9.25) mm, rotated rx 180 ry 0 rz 90 deg; joints [70.718, -18.26, 87.83, 0, 20.43, 70.718] to (-72.01, -72.95, -9.25) mm, rotated rx 180 ry 0 rz 90 deg; joints [70.695, -18.232, 87.713, 0, 20.519, 70.695]
  MoveC 6158 to (-71.33, -73.19, -9.25) mm, rotated rx -180 ry 0 rz 90 deg; joints [70.695, -18.22, 87.661, 0, 20.559, 70.695] to (-70.6, -73.27, -9.25) mm, rotated rx -180 ry 0 rz 90 deg; joints [70.7, -18.208, 87.61, 0, 20.598, 70.7]
  MoveL 6159 to (-43.12, -73, -9.25) mm, rotated rx -180 ry 0 rz 90 deg; joints [71.018, -17.755, 85.748, 0, 22.007, 71.018]
  MoveL 6160 to (-35.83, -72.92, -9.25) mm, rotated rx 180 ry 0 rz 90 deg; joints [71.101, -17.629, 85.248, 0, 22.381, 71.101]
  MoveC 6161 to (-33.92, -72.21, -9.25) mm, rotated rx 180 ry 0 rz 90 deg; joints [71.145, -17.6, 85.133, 0, 22.467, 71.145] to (-32.82, -70.5, -9.25) mm, rotated rx -180 ry 0 rz 90 deg; joints [71.212, -17.591, 85.096, 0, 22.494, 71.212]
  MoveL 6162 to (-26.79, -47.32, -9.25) mm, rotated rx 180 ry 0 rz 90 deg; joints [72.021, -17.62, 85.213, 0, 22.407, 72.021]
  MoveL 6163 to (-34.1, -45.42, -9.25) mm, rotated rx -180 ry 0 rz 90 deg; joints [72.006, -17.758, 85.762, 0, 21.996, 72.006]
  MoveL 6164 to (-34.1, -45.42, -6.25) mm, rotated rx -180 ry 0 rz 90 deg; joints [72.006, -17.913, 85.864, 0, 22.049, 72.006]
  Establecer velocidad (1000.0 mm/s)
  MoveL 6165 to (-34.1, -45.42, 10) mm, rotated rx 180 ry 0 rz 90 deg; joints [72.006, -18.748, 86.407, 0, 22.341, 72.006]
  Establecer velocidad (66.7 mm/s)
  MoveL 6166 to (-65.59, 36.24, 10) mm, rotated rx 180 ry 0 rz 90 deg; joints [74.396, -19.67, 90.235, 0, 19.435, 74.396]
  MoveL 6167 to (-65.59, 36.24, -6) mm, rotated rx 180 ry 0 rz 90 deg; joints [74.396, -18.833, 89.7, 0, 19.133, 74.396]
  MoveL 6168 to (-67.09, 36.43, -6.41) mm, rotated rx 180 ry 0 rz 90 deg; joints [74.388, -18.835, 89.791, 0, 19.044, 74.388]
  MoveL 6169 to (-68.6, 36.25, -6.81) mm, rotated rx -180 ry 0 rz 90 deg; joints [74.368, -18.835, 89.875, 0, 18.96, 74.368]
  MoveL 6170 to (-70.03, 35.74, -7.22) mm, rotated rx -180 ry 0 rz 90 deg; joints [74.337, -18.833, 89.948, 0, 18.886, 74.337]
  MoveL 6171 to (-71.31, 34.92, -7.63) mm, rotated rx -180 ry 0 rz 90 deg; joints [74.297, -18.827, 90.004, 0, 18.823, 74.297]
  MoveL 6172 to (-72.38, 33.84, -8.03) mm, rotated rx -180 ry 0 rz 90 deg; joints [74.25, -18.817, 90.042, 0, 18.776, 74.25]
  MoveL 6173 to (-73.19, 32.55, -8.44) mm, rotated rx 180 ry 0 rz 90 deg; joints [74.199, -18.802, 90.057, 0, 18.745, 74.199]
  MoveL 6174 to (-73.69, 31.12, -8.84) mm, rotated rx 180 ry 0 rz 90 deg; joints [74.145, -18.782, 90.05, 0, 18.733, 74.145]
  MoveL 6175 to (-73.83, 29.6, -9.25) mm, rotated rx 180 ry 0 rz 90 deg; joints [74.092, -18.757, 90.016, 0, 18.74, 74.092]
  MoveL 6176 to (-73.83, 1.85, -9.25) mm, rotated rx 180 ry 0 rz 90 deg; joints [73.155, -18.636, 89.471, 0, 19.165, 73.155]
  MoveC 6177 to (-73.76, 1.15, -9.25) mm, rotated rx 180 ry 0 rz 90 deg; joints [73.132, -18.632, 89.453, 0, 19.179, 73.132] to (-73.57, 0.47, -9.25) mm, rotated rx 180 ry 0 rz 90 deg; joints [73.111, -18.626, 89.427, 0, 19.2, 73.111]
  MoveC 6178 to (-72.68, -0.7, -9.25) mm, rotated rx -180 ry 0 rz 90 deg; joints [73.081, -18.608, 89.343, 0, 19.265, 73.081] to (-71.39, -1.41, -9.25) mm, rotated rx -180 ry 0 rz 90 deg; joints [73.07, -18.585, 89.242, 0, 19.343, 73.07]
  MoveC 6179 to (-70.72, -1.53, -9.25) mm, rotated rx 180 ry 0 rz 90 deg; joints [73.073, -18.574, 89.195, 0, 19.38, 73.073] to (-70.05, -1.46, -9.25) mm, rotated rx -180 ry 0 rz 90 deg; joints [73.082, -18.564, 89.151, 0, 19.414, 73.082]
  MoveL 6180 to (-63.02, 0.14, -9.25) mm, rotated rx 180 ry 0 rz 90 deg; joints [73.207, -18.465, 88.711, 0, 19.754, 73.207]
  MoveL 6181 to (-27.01, 8.51, -9.25) mm, rotated rx -180 ry 0 rz 90 deg; joints [73.837, -17.921, 86.419, 0, 21.502, 73.837]
  MoveL 6182 to (-22.27, 9.63, -9.25) mm, rotated rx 180 ry 0 rz 90 deg; joints [73.919, -17.845, 86.112, 0, 21.733, 73.919]
  MoveC 6183 to (-21.22, 10.09, -9.25) mm, rotated rx 180 ry 0 rz 90 deg; joints [73.944, -17.83, 86.048, 0, 21.781, 73.944] to (-20.42, 10.9, -9.25) mm, rotated rx 180 ry 0 rz 90 deg; joints [73.978, -17.82, 86.009, 0, 21.811, 73.978]
  MoveC 6184 to (-19.77, 12.36, -9.25) mm, rotated rx 180 ry 0 rz 90 deg; joints [74.032, -17.816, 85.993, 0, 21.823, 74.032] to (-19.9, 13.95, -9.25) mm, rotated rx -180 ry 0 rz 90 deg; joints [74.083, -17.826, 86.033, 0, 21.793, 74.083]
  MoveL 6185 to (-20.14, 14.69, -9.25) mm, rotated rx -180 ry 0 rz 90 deg; joints [74.105, -17.834, 86.065, 0, 21.769, 74.105]
  MoveL 6186 to (-26.06, 31.26, -9.25) mm, rotated rx -180 ry 0 rz 90 deg; joints [74.597, -18.013, 86.799, 0, 21.215, 74.597]
  MoveL 6187 to (-26.25, 31.75, -9.25) mm, rotated rx -180 ry 0 rz 90 deg; joints [74.611, -18.019, 86.821, 0, 21.198, 74.611]
  MoveL 6188 to (-26.81, 32.69, -9.25) mm, rotated rx 180 ry 0 rz 90 deg; joints [74.637, -18.033, 86.878, 0, 21.155, 74.637]
  MoveC 6189 to (-27.13, 33.02, -9.25) mm, rotated rx -180 ry 0 rz 90 deg; joints [74.645, -18.04, 86.906, 0, 21.133, 74.645] to (-27.49, 33.3, -9.25) mm, rotated rx 180 ry 0 rz 90 deg; joints [74.651, -18.047, 86.936, 0, 21.11, 74.651]
  MoveL 6190 to (-63.97, 56.77, -9.25) mm, rotated rx -180 ry 0 rz 90 deg; joints [75.109, -18.722, 89.857, 0, 18.865, 75.109]
  MoveL 6191 to (-69.29, 60.18, -9.25) mm, rotated rx 180 ry 0 rz 90 deg; joints [75.177, -18.813, 90.275, 0, 18.538, 75.177]
  MoveC 6192 to (-71.19, 60.17, -9.25) mm, rotated rx -180 ry 0 rz 90 deg; joints [75.159, -18.841, 90.402, 0, 18.439, 75.159] to (-72.83, 59.23, -9.25) mm, rotated rx 180 ry 0 rz 90 deg; joints [75.112, -18.861, 90.495, 0, 18.366, 75.112]
  MoveL 6193 to (-73.34, 58.65, -9.25) mm, rotated rx -180 ry 0 rz 90 deg; joints [75.088, -18.866, 90.519, 0, 18.347, 75.088]
  MoveC 6194 to (-73.7, 58.05, -9.25) mm, rotated rx -180 ry 0 rz 90 deg; joints [75.064, -18.869, 90.532, 0, 18.337, 75.064] to (-73.83, 57.36, -9.25) mm, rotated rx 180 ry 0 rz 90 deg; joints [75.039, -18.868, 90.528, 0, 18.34, 75.039]
  MoveL 6195 to (-73.83, 29.6, -9.25) mm, rotated rx 180 ry 0 rz 90 deg; joints [74.092, -18.757, 90.016, 0, 18.74, 74.092]
  MoveL 6196 to (-66.27, 29.6, -9.25) mm, rotated rx -180 ry 0 rz 90 deg; joints [74.165, -18.645, 89.511, 0, 19.135, 74.165]
  MoveL 6197 to (-66.27, 29.6, -6.25) mm, rotated rx -180 ry 0 rz 90 deg; joints [74.165, -18.802, 89.612, 0, 19.19, 74.165]
  Establecer velocidad (1000.0 mm/s)
  MoveL 6198 to (-66.27, 29.6, 10) mm, rotated rx -180 ry 0 rz 90 deg; joints [74.165, -19.652, 90.156, 0, 19.496, 74.165]
  Establecer velocidad (66.7 mm/s)
  MoveL 6199 to (-65.42, 36.24, 10) mm, rotated rx 180 ry 0 rz 90 deg; joints [74.398, -19.667, 90.224, 0, 19.444, 74.398]
  MoveL 6200 to (-65.42, 36.24, -6.25) mm, rotated rx -180 ry 0 rz 90 deg; joints [74.398, -18.817, 89.681, 0, 19.137, 74.398]
  MoveL 6201 to (-66.93, 36.43, -6.66) mm, rotated rx 180 ry 0 rz 90 deg; joints [74.39, -18.819, 89.771, 0, 19.048, 74.39]
  MoveL 6202 to (-68.44, 36.25, -7.06) mm, rotated rx 180 ry 0 rz 90 deg; joints [74.37, -18.82, 89.855, 0, 18.964, 74.37]
  MoveL 6203 to (-69.87, 35.74, -7.47) mm, rotated rx 180 ry 0 rz 90 deg; joints [74.339, -18.818, 89.928, 0, 18.89, 74.339]
  MoveL 6204 to (-71.15, 34.92, -7.87) mm, rotated rx -180 ry 0 rz 90 deg; joints [74.299, -18.812, 89.985, 0, 18.827, 74.299]
  MoveL 6205 to (-72.22, 33.84, -8.28) mm, rotated rx 180 ry 0 rz 90 deg; joints [74.252, -18.802, 90.022, 0, 18.78, 74.252]
  MoveL 6206 to (-73.02, 32.55, -8.69) mm, rotated rx 180 ry 0 rz 90 deg; joints [74.2, -18.787, 90.038, 0, 18.749, 74.2]
  MoveL 6207 to (-73.52, 31.12, -9.09) mm, rotated rx -180 ry 0 rz 90 deg; joints [74.147, -18.767, 90.03, 0, 18.737, 74.147]
  MoveL 6208 to (-73.66, 29.6, -9.5) mm, rotated rx 180 ry 0 rz 90 deg; joints [74.094, -18.741, 89.997, 0, 18.745, 74.094]
  MoveL 6209 to (-73.66, 2.37, -9.5) mm, rotated rx -180 ry 0 rz 90 deg; joints [73.174, -18.623, 89.462, 0, 19.161, 73.174]
  MoveL 6210 to (-73.63, 1.42, -9.5) mm, rotated rx 180 ry 0 rz 90 deg; joints [73.142, -18.618, 89.441, 0, 19.178, 73.142]
  MoveC 6211 to (-72.42, -0.64, -9.5) mm, rotated rx -180 ry 0 rz 90 deg; joints [73.085, -18.591, 89.318, 0, 19.273, 73.085] to (-70.13, -1.33, -9.5) mm, rotated rx 180 ry 0 rz 90 deg; joints [73.086, -18.553, 89.151, 0, 19.403, 73.086]
  MoveL 6212 to (-63.02, 0.29, -9.5) mm, rotated rx 180 ry 0 rz 90 deg; joints [73.212, -18.452, 88.706, 0, 19.747, 73.212]
  MoveL 6213 to (-27.01, 8.68, -9.5) mm, rotated rx -180 ry 0 rz 90 deg; joints [73.843, -17.909, 86.414, 0, 21.495, 73.843]
  MoveL 6214 to (-22.4, 9.79, -9.5) mm, rotated rx -180 ry 0 rz 90 deg; joints [73.923, -17.835, 86.116, 0, 21.72, 73.923]
  MoveC 6215 to (-21.2, 10.38, -9.5) mm, rotated rx 180 ry 0 rz 90 deg; joints [73.954, -17.818, 86.044, 0, 21.774, 73.954] to (-20.37, 11.45, -9.5) mm, rotated rx 180 ry 0 rz 90 deg; joints [73.996, -17.809, 86.008, 0, 21.801, 73.996]
  MoveC 6216 to (-19.94, 12.67, -9.5) mm, rotated rx -180 ry 0 rz 90 deg; joints [74.041, -17.807, 86.002, 0, 21.805, 74.041] to (-20.07, 13.96, -9.5) mm, rotated rx 180 ry 0 rz 90 deg; joints [74.082, -17.816, 86.037, 0, 21.779, 74.082]
  MoveL 6217 to (-20.31, 14.69, -9.5) mm, rotated rx 180 ry 0 rz 90 deg; joints [74.103, -17.824, 86.068, 0, 21.756, 74.103]
  MoveL 6218 to (-26.06, 30.8, -9.5) mm, rotated rx -180 ry 0 rz 90 deg; joints [74.581, -17.998, 86.781, 0, 21.217, 74.581]
  MoveL 6219 to (-26.42, 31.75, -9.5) mm, rotated rx 180 ry 0 rz 90 deg; joints [74.61, -18.009, 86.824, 0, 21.185, 74.61]
  MoveL 6220 to (-27.02, 32.69, -9.5) mm, rotated rx -180 ry 0 rz 90 deg; joints [74.635, -18.023, 86.884, 0, 21.139, 74.635]
  MoveC 6221 to (-27.66, 33.19, -9.5) mm, rotated rx -180 ry 0 rz 90 deg; joints [74.646, -18.036, 86.937, 0, 21.099, 74.646] to (-28.32, 33.64, -9.5) mm, rotated rx 180 ry 0 rz 90 deg; joints [74.655, -18.049, 86.992, 0, 21.057, 74.655]
  MoveL 6222 to (-63.97, 56.6, -9.5) mm, rotated rx -180 ry 0 rz 90 deg; joints [75.103, -18.708, 89.846, 0, 18.862, 75.103]
  MoveL 6223 to (-69.18, 59.94, -9.5) mm, rotated rx -180 ry 0 rz 90 deg; joints [75.17, -18.798, 90.255, 0, 18.543, 75.17]
  MoveC 6224 to (-71.63, 59.71, -9.5) mm, rotated rx 180 ry 0 rz 90 deg; joints [75.14, -18.832, 90.415, 0, 18.417, 75.14] to (-73.44, 58.03, -9.5) mm, rotated rx 180 ry 0 rz 90 deg; joints [75.066, -18.852, 90.506, 0, 18.346, 75.066]
  MoveC 6225 to (-73.6, 57.6, -9.5) mm, rotated rx -180 ry 0 rz 90 deg; joints [75.049, -18.853, 90.509, 0, 18.343, 75.049] to (-73.66, 57.14, -9.5) mm, rotated rx 180 ry 0 rz 90 deg; joints [75.033, -18.852, 90.505, 0, 18.347, 75.033]
  MoveL 6226 to (-73.66, 29.6, -9.5) mm, rotated rx 180 ry 0 rz 90 deg; joints [74.094, -18.741, 89.997, 0, 18.745, 74.094]
  MoveL 6227 to (-66.11, 29.6, -9.5) mm, rotated rx 180 ry 0 rz 90 deg; joints [74.167, -18.63, 89.491, 0, 19.139, 74.167]
  MoveL 6228 to (-66.11, 29.6, -6.5) mm, rotated rx 180 ry 0 rz 90 deg; joints [74.167, -18.787, 89.593, 0, 19.194, 74.167]
  Establecer velocidad (1000.0 mm/s)
  MoveL 6229 to (-66.11, 29.6, 10) mm, rotated rx -180 ry 0 rz 90 deg; joints [74.167, -19.649, 90.145, 0, 19.505, 74.167]
  Establecer velocidad (66.7 mm/s)
  MoveL 6230 to (-39.77, -31.86, 10) mm, rotated rx 180 ry 0 rz 90 deg; joints [72.388, -18.922, 87.098, 0, 21.824, 72.388]
  MoveL 6231 to (-39.77, -31.86, -6.25) mm, rotated rx 180 ry 0 rz 90 deg; joints [72.388, -18.084, 86.555, 0, 21.529, 72.388]
  MoveL 6232 to (-39.9, -30.35, -6.66) mm, rotated rx 180 ry 0 rz 90 deg; joints [72.436, -18.073, 86.583, 0, 21.49, 72.436]
  MoveL 6233 to (-40.38, -28.91, -7.06) mm, rotated rx 180 ry 0 rz 90 deg; joints [72.478, -18.068, 86.634, 0, 21.434, 72.478]
  MoveL 6234 to (-41.18, -27.61, -7.47) mm, rotated rx 180 ry 0 rz 90 deg; joints [72.512, -18.068, 86.703, 0, 21.364, 72.512]
  MoveL 6235 to (-42.24, -26.52, -7.87) mm, rotated rx -180 ry 0 rz 90 deg; joints [72.537, -18.07, 86.786, 0, 21.284, 72.537]
  MoveL 6236 to (-43.52, -25.7, -8.28) mm, rotated rx -180 ry 0 rz 90 deg; joints [72.551, -18.075, 86.877, 0, 21.198, 72.551]
  MoveL 6237 to (-44.94, -25.17, -8.69) mm, rotated rx 180 ry 0 rz 90 deg; joints [72.553, -18.08, 86.972, 0, 21.108, 72.553]
  MoveL 6238 to (-46.45, -24.98, -9.09) mm, rotated rx -180 ry 0 rz 90 deg; joints [72.544, -18.085, 87.066, 0, 21.019, 72.544]
  MoveL 6239 to (-47.96, -25.15, -9.5) mm, rotated rx -180 ry 0 rz 90 deg; joints [72.523, -18.088, 87.151, 0, 20.937, 72.523]
  MoveC 6240 to (-59.54, -27.59, -9.5) mm, rotated rx -180 ry 0 rz 90 deg; joints [72.321, -18.262, 87.886, 0, 20.376, 72.321] to (-71.12, -30.04, -9.5) mm, rotated rx 180 ry 0 rz 90 deg; joints [72.118, -18.431, 88.614, 0, 19.817, 72.118]
  MoveC 6241 to (-72.07, -30.38, -9.5) mm, rotated rx -180 ry 0 rz 90 deg; joints [72.096, -18.444, 88.67, 0, 19.774, 72.096] to (-72.86, -31.01, -9.5) mm, rotated rx 180 ry 0 rz 90 deg; joints [72.067, -18.453, 88.709, 0, 19.744, 72.067]
  MoveC 6242 to (-73.45, -31.98, -9.5) mm, rotated rx 180 ry 0 rz 90 deg; joints [72.028, -18.457, 88.728, 0, 19.729, 72.028] to (-73.66, -33.1, -9.5) mm, rotated rx -180 ry 0 rz 90 deg; joints [71.988, -18.455, 88.717, 0, 19.738, 71.988]
  MoveL 6243 to (-73.66, -69.95, -9.5) mm, rotated rx -180 ry 0 rz 90 deg; joints [70.774, -18.262, 87.885, 0, 20.377, 70.774]
  MoveC 6244 to (-72.72, -72.2, -9.5) mm, rotated rx 180 ry 0 rz 90 deg; joints [70.711, -18.235, 87.77, 0, 20.465, 70.711] to (-70.46, -73.12, -9.5) mm, rotated rx -180 ry 0 rz 90 deg; joints [70.707, -18.194, 87.596, 0, 20.598, 70.707]
  MoveL 6245 to (-69.65, -73.11, -9.5) mm, rotated rx -180 ry 0 rz 90 deg; joints [70.716, -18.181, 87.542, 0, 20.639, 70.716]
  MoveL 6246 to (-35.96, -72.76, -9.5) mm, rotated rx -180 ry 0 rz 90 deg; joints [71.105, -17.619, 85.252, 0, 22.368, 71.105]
  MoveC 6247 to (-34.51, -72.38, -9.5) mm, rotated rx 180 ry 0 rz 90 deg; joints [71.133, -17.596, 85.161, 0, 22.436, 71.133] to (-33.41, -71.38, -9.5) mm, rotated rx -180 ry 0 rz 90 deg; joints [71.177, -17.583, 85.108, 0, 22.475, 71.177]
  MoveC 6248 to (-33.18, -71.01, -9.5) mm, rotated rx -180 ry 0 rz 90 deg; joints [71.192, -17.581, 85.101, 0, 22.48, 71.192] to (-33.01, -70.6, -9.5) mm, rotated rx 180 ry 0 rz 90 deg; joints [71.206, -17.581, 85.099, 0, 22.482, 71.206]
  MoveL 6249 to (-32.75, -69.65, -9.5) mm, rotated rx 180 ry 0 rz 90 deg; joints [71.24, -17.582, 85.103, 0, 22.478, 71.24]
  MoveL 6250 to (-21.06, -24.64, -9.5) mm, rotated rx 180 ry 0 rz 90 deg; joints [72.813, -17.633, 85.306, 0, 22.327, 72.813]
  MoveC 6251 to (-20.96, -24.17, -9.5) mm, rotated rx -180 ry 0 rz 90 deg; joints [72.83, -17.634, 85.309, 0, 22.325, 72.83] to (-20.93, -23.69, -9.5) mm, rotated rx 180 ry 0 rz 90 deg; joints [72.845, -17.636, 85.317, 0, 22.319, 72.845]
  MoveC 6252 to (-21.35, -22.43, -9.5) mm, rotated rx -180 ry 0 rz 90 deg; joints [72.882, -17.65, 85.373, 0, 22.277, 72.882] to (-23.22, -20.59, -9.5) mm, rotated rx 180 ry 0 rz 90 deg; joints [72.923, -17.693, 85.543, 0, 22.15, 72.923]
  MoveL 6253 to (-23.63, -20.42, -9.5) mm, rotated rx -180 ry 0 rz 90 deg; joints [72.924, -17.701, 85.576, 0, 22.125, 72.924]
  MoveC 6254 to (-24.2, -20.29, -9.5) mm, rotated rx 180 ry 0 rz 90 deg; joints [72.923, -17.712, 85.618, 0, 22.094, 72.923] to (-24.78, -20.32, -9.5) mm, rotated rx 180 ry 0 rz 90 deg; joints [72.916, -17.722, 85.658, 0, 22.064, 72.916]
  MoveC 6255 to (-36.37, -22.73, -9.5) mm, rotated rx -180 ry 0 rz 90 deg; joints [72.721, -17.908, 86.408, 0, 21.499, 72.721] to (-47.96, -25.15, -9.5) mm, rotated rx 180 ry 0 rz 90 deg; joints [72.523, -18.088, 87.151, 0, 20.937, 72.523]
  MoveL 6256 to (-46.41, -32.54, -9.5) mm, rotated rx 180 ry 0 rz 90 deg; joints [72.296, -18.024, 86.885, 0, 21.138, 72.296]
  MoveL 6257 to (-46.41, -32.54, -6.5) mm, rotated rx 180 ry 0 rz 90 deg; joints [72.296, -18.179, 86.987, 0, 21.192, 72.296]
  Establecer velocidad (1000.0 mm/s)
  MoveL 6258 to (-46.41, -32.54, 10) mm, rotated rx 180 ry 0 rz 90 deg; joints [72.296, -19.031, 87.538, 0, 21.493, 72.296]
  Establecer velocidad (66.7 mm/s)
  MoveL 6259 to (15.52, -63.96, 10) mm, rotated rx 180 ry 0 rz 90 deg; joints [71.93, -17.702, 82.48, 0, 25.223, 71.93]
  MoveL 6260 to (15.52, -63.96, -6.25) mm, rotated rx 180 ry 0 rz 90 deg; joints [71.93, -16.88, 81.935, 0, 24.945, 71.93]
  MoveL 6261 to (15.38, -65.47, -6.66) mm, rotated rx 180 ry 0 rz 90 deg; joints [71.881, -16.852, 81.896, 0, 24.957, 71.881]
  MoveL 6262 to (15.6, -66.97, -7.06) mm, rotated rx 180 ry 0 rz 90 deg; joints [71.836, -16.817, 81.83, 0, 24.987, 71.836]
  MoveL 6263 to (16.15, -68.39, -7.47) mm, rotated rx -180 ry 0 rz 90 deg; joints [71.798, -16.777, 81.743, 0, 25.034, 71.798]
  MoveL 6264 to (17.01, -69.65, -7.87) mm, rotated rx 180 ry 0 rz 90 deg; joints [71.767, -16.731, 81.637, 0, 25.093, 71.767]
  MoveL 6265 to (18.12, -70.69, -8.28) mm, rotated rx 180 ry 0 rz 90 deg; joints [71.746, -16.681, 81.519, 0, 25.163, 71.746]
  MoveL 6266 to (19.43, -71.45, -8.69) mm, rotated rx -180 ry 0 rz 90 deg; joints [71.736, -16.629, 81.391, 0, 25.238, 71.736]
  MoveL 6267 to (20.88, -71.91, -9.09) mm, rotated rx -180 ry 0 rz 90 deg; joints [71.736, -16.576, 81.262, 0, 25.315, 71.736]
  MoveL 6268 to (22.39, -72.01, -9.5) mm, rotated rx -180 ry 0 rz 90 deg; joints [71.749, -16.525, 81.135, 0, 25.389, 71.749]
  MoveC 6269 to (33.14, -71.67, -9.5) mm, rotated rx -180 ry 0 rz 90 deg; joints [71.869, -16.307, 80.359, 0, 25.948, 71.869] to (43.89, -71.28, -9.5) mm, rotated rx -180 ry 0 rz 90 deg; joints [71.99, -16.084, 79.576, 0, 26.508, 71.99]
  MoveC 6270 to (46.24, -68.33, -9.5) mm, rotated rx -180 ry 0 rz 90 deg; joints [72.104, -16.054, 79.473, 0, 26.582, 72.104] to (46.38, -64.56, -9.5) mm, rotated rx -180 ry 0 rz 90 deg; joints [72.222, -16.077, 79.552, 0, 26.525, 72.222]
  MoveC 6271 to (35.33, -51.21, -9.5) mm, rotated rx 180 ry 0 rz 90 deg; joints [72.528, -16.397, 80.68, 0, 25.717, 72.528] to (24.17, -37.97, -9.5) mm, rotated rx -180 ry 0 rz 90 deg; joints [72.834, -16.707, 81.796, 0, 24.912, 72.834]
  MoveL 6272 to (23.57, -37.43, -9.5) mm, rotated rx 180 ry 0 rz 90 deg; joints [72.845, -16.722, 81.851, 0, 24.871, 72.845]
  MoveL 6273 to (17.74, -32.69, -9.5) mm, rotated rx -180 ry 0 rz 90 deg; joints [72.938, -16.866, 82.378, 0, 24.488, 72.938]
  MoveL 6274 to (13.08, -28.9, -9.5) mm, rotated rx 180 ry 0 rz 90 deg; joints [73.013, -16.979, 82.797, 0, 24.182, 73.013]
  MoveC 6275 to (10.45, -28.36, -9.5) mm, rotated rx 180 ry 0 rz 90 deg; joints [73.005, -17.033, 82.997, 0, 24.036, 73.005] to (8.05, -29.56, -9.5) mm, rotated rx 180 ry 0 rz 90 deg; joints [72.943, -17.071, 83.142, 0, 23.929, 72.943]
  MoveC 6276 to (7.75, -29.97, -9.5) mm, rotated rx -180 ry 0 rz 90 deg; joints [72.927, -17.075, 83.155, 0, 23.919, 72.927] to (7.55, -30.44, -9.5) mm, rotated rx -180 ry 0 rz 90 deg; joints [72.91, -17.076, 83.159, 0, 23.917, 72.91]
  MoveL 6277 to (5.68, -37.43, -9.5) mm, rotated rx 180 ry 0 rz 90 deg; joints [72.669, -17.07, 83.138, 0, 23.932, 72.669]
  MoveL 6278 to (-2.58, -68.07, -9.5) mm, rotated rx 180 ry 0 rz 90 deg; joints [71.613, -17.04, 83.023, 0, 24.016, 71.613]
  MoveC 6279 to (-1.96, -71.15, -9.5) mm, rotated rx 180 ry 0 rz 90 deg; joints [71.522, -17.008, 82.906, 0, 24.102, 71.522] to (0.88, -72.5, -9.5) mm, rotated rx 180 ry 0 rz 90 deg; joints [71.509, -16.945, 82.672, 0, 24.274, 71.509]
  MoveC 6280 to (11.64, -72.28, -9.5) mm, rotated rx -180 ry 0 rz 90 deg; joints [71.629, -16.738, 81.906, 0, 24.831, 71.629] to (22.39, -72.01, -9.5) mm, rotated rx -180 ry 0 rz 90 deg; joints [71.749, -16.525, 81.135, 0, 25.389, 71.749]
  MoveL 6281 to (22.17, -64.46, -9.5) mm, rotated rx 180 ry 0 rz 90 deg; joints [71.982, -16.579, 81.331, 0, 25.248, 71.982]
  MoveL 6282 to (22.17, -64.46, -6.5) mm, rotated rx 180 ry 0 rz 90 deg; joints [71.982, -16.731, 81.433, 0, 25.298, 71.982]
  Establecer velocidad (1000.0 mm/s)
  MoveL 6283 to (22.17, -64.46, 10) mm, rotated rx 180 ry 0 rz 90 deg; joints [71.982, -17.565, 81.987, 0, 25.578, 71.982]
  Establecer velocidad (66.7 mm/s)
  MoveL 6284 to (59.71, -30.02, 10) mm, rotated rx -180 ry 0 rz 90 deg; joints [73.42, -16.999, 80.014, 0, 26.986, 73.42]
  MoveL 6285 to (59.71, -30.02, -6.25) mm, rotated rx 180 ry 0 rz 90 deg; joints [73.42, -16.184, 79.466, 0, 26.718, 73.42]
  MoveL 6286 to (62.53, -33.13, -7.38) mm, rotated rx -180 ry 0 rz 90 deg; joints [73.35, -16.046, 79.147, 0, 26.899, 73.35]
  MoveL 6287 to (62.53, -25.21, -9.5) mm, rotated rx -180 ry 0 rz 90 deg; joints [73.596, -15.99, 79.25, 0, 26.74, 73.596]
  MoveL 6288 to (62.53, -17.28, -9.5) mm, rotated rx 180 ry 0 rz 90 deg; joints [73.842, -16.04, 79.423, 0, 26.617, 73.842]
  MoveL 6289 to (57.56, -23.97, -9.5) mm, rotated rx -180 ry 0 rz 90 deg; joints [73.589, -16.105, 79.649, 0, 26.456, 73.589]
  MoveC 6290 to (56.96, -25.96, -9.5) mm, rotated rx 180 ry 0 rz 90 deg; joints [73.521, -16.105, 79.65, 0, 26.455, 73.521] to (57.76, -27.87, -9.5) mm, rotated rx 180 ry 0 rz 90 deg; joints [73.469, -16.076, 79.548, 0, 26.528, 73.469]
  MoveL 6291 to (58.71, -28.9, -9.5) mm, rotated rx -180 ry 0 rz 90 deg; joints [73.446, -16.049, 79.455, 0, 26.594, 73.446]
  MoveL 6292 to (62.53, -33.13, -9.5) mm, rotated rx -180 ry 0 rz 90 deg; joints [73.35, -15.939, 79.074, 0, 26.865, 73.35]
  MoveL 6293 to (62.53, -25.21, -9.5) mm, rotated rx -180 ry 0 rz 90 deg; joints [73.596, -15.99, 79.25, 0, 26.74, 73.596]
  MoveL 6294 to (62.53, -17.66, -9.5) mm, rotated rx 180 ry 0 rz 90 deg; joints [73.83, -16.038, 79.415, 0, 26.622, 73.83]
  MoveL 6295 to (62.53, -17.66, -6.5) mm, rotated rx -180 ry 0 rz 90 deg; joints [73.83, -16.189, 79.518, 0, 26.671, 73.83]
  Establecer velocidad (1000.0 mm/s)
  MoveL 6296 to (62.53, -17.66, 10) mm, rotated rx -180 ry 0 rz 90 deg; joints [73.83, -17.017, 80.074, 0, 26.943, 73.83]
  Establecer velocidad (66.7 mm/s)
  MoveL 6297 to (35.34, 19.15, 10) mm, rotated rx -180 ry 0 rz 90 deg; joints [74.75, -17.804, 82.846, 0, 24.958, 74.75]
  MoveL 6298 to (35.34, 19.15, -6.25) mm, rotated rx 180 ry 0 rz 90 deg; joints [74.75, -16.98, 82.301, 0, 24.679, 74.75]
  MoveL 6299 to (35.51, 20.66, -6.66) mm, rotated rx -180 ry 0 rz 90 deg; joints [74.8, -16.964, 82.305, 0, 24.659, 74.8]
  MoveL 6300 to (35.32, 22.17, -7.06) mm, rotated rx -180 ry 0 rz 90 deg; joints [74.846, -16.955, 82.335, 0, 24.621, 74.846]
  MoveL 6301 to (34.8, 23.59, -7.47) mm, rotated rx 180 ry 0 rz 90 deg; joints [74.887, -16.953, 82.387, 0, 24.566, 74.887]
  MoveL 6302 to (33.97, 24.87, -7.87) mm, rotated rx -180 ry 0 rz 90 deg; joints [74.921, -16.955, 82.459, 0, 24.497, 74.921]
  MoveL 6303 to (32.88, 25.93, -8.28) mm, rotated rx 180 ry 0 rz 90 deg; joints [74.946, -16.962, 82.545, 0, 24.417, 74.946]
  MoveL 6304 to (31.59, 26.73, -8.69) mm, rotated rx -180 ry 0 rz 90 deg; joints [74.96, -16.971, 82.641, 0, 24.33, 74.96]
  MoveL 6305 to (30.15, 27.22, -9.09) mm, rotated rx -180 ry 0 rz 90 deg; joints [74.963, -16.981, 82.741, 0, 24.24, 74.963]
  MoveL 6306 to (28.64, 27.34, -9.5) mm, rotated rx 180 ry 0 rz 90 deg; joints [74.954, -16.99, 82.839, 0, 24.151, 74.954]
  MoveC 6307 to (20.71, 27.27, -9.5) mm, rotated rx -180 ry 0 rz 90 deg; joints [74.883, -17.142, 83.41, 0, 23.733, 74.883] to (12.79, 27.17, -9.5) mm, rotated rx 180 ry 0 rz 90 deg; joints [74.811, -17.291, 83.976, 0, 23.315, 74.811]
  MoveL 6308 to (11.85, 27.09, -9.5) mm, rotated rx 180 ry 0 rz 90 deg; joints [74.8, -17.309, 84.043, 0, 23.266, 74.8]
  MoveC 6309 to (9.63, 25.57, -9.5) mm, rotated rx 180 ry 0 rz 90 deg; joints [74.731, -17.342, 84.171, 0, 23.171, 74.731] to (9, 22.96, -9.5) mm, rotated rx 180 ry 0 rz 90 deg; joints [74.641, -17.341, 84.165, 0, 23.176, 74.641]
  MoveL 6310 to (9.07, 22.74, -9.5) mm, rotated rx -180 ry 0 rz 90 deg; joints [74.634, -17.338, 84.156, 0, 23.182, 74.634]
  MoveL 6311 to (13.06, 11.85, -9.5) mm, rotated rx 180 ry 0 rz 90 deg; joints [74.318, -17.207, 83.655, 0, 23.552, 74.318]
  MoveL 6312 to (13.41, 10.9, -9.5) mm, rotated rx 180 ry 0 rz 90 deg; joints [74.291, -17.195, 83.61, 0, 23.585, 74.291]
  MoveL 6313 to (13.74, 10.14, -9.5) mm, rotated rx -180 ry 0 rz 90 deg; joints [74.269, -17.185, 83.571, 0, 23.614, 74.269]
  MoveC 6314 to (14.18, 9.51, -9.5) mm, rotated rx -180 ry 0 rz 90 deg; joints [74.253, -17.174, 83.527, 0, 23.646, 74.253] to (14.74, 9, -9.5) mm, rotated rx -180 ry 0 rz 90 deg; joints [74.242, -17.16, 83.476, 0, 23.684, 74.242]
  MoveL 6315 to (28.39, -1.29, -9.5) mm, rotated rx -180 ry 0 rz 90 deg; joints [74.036, -16.84, 82.281, 0, 24.559, 74.036]
  MoveC 6316 to (29.06, -1.67, -9.5) mm, rotated rx -180 ry 0 rz 90 deg; joints [74.03, -16.824, 82.224, 0, 24.6, 74.03] to (29.81, -1.84, -9.5) mm, rotated rx 180 ry 0 rz 90 deg; joints [74.032, -16.808, 82.166, 0, 24.642, 74.032]
  MoveC 6317 to (31.98, -1.44, -9.5) mm, rotated rx 180 ry 0 rz 90 deg; joints [74.064, -16.768, 82.017, 0, 24.751, 74.064] to (33.64, -0.01, -9.5) mm, rotated rx 180 ry 0 rz 90 deg; joints [74.125, -16.743, 81.925, 0, 24.817, 74.125]
  MoveL 6318 to (47.18, 19.43, -9.5) mm, rotated rx -180 ry 0 rz 90 deg; joints [74.861, -16.578, 81.328, 0, 25.25, 74.861]
  MoveL 6319 to (48.23, 20.99, -9.5) mm, rotated rx 180 ry 0 rz 90 deg; joints [74.92, -16.565, 81.282, 0, 25.283, 74.92]
  MoveC 6320 to (47.89, 24.65, -9.5) mm, rotated rx -180 ry 0 rz 90 deg; joints [75.033, -16.593, 81.38, 0, 25.213, 75.033] to (45.43, 27.4, -9.5) mm, rotated rx 180 ry 0 rz 90 deg; joints [75.1, -16.657, 81.614, 0, 25.043, 75.1]
  MoveC 6321 to (37.03, 27.39, -9.5) mm, rotated rx 180 ry 0 rz 90 deg; joints [75.028, -16.826, 82.229, 0, 24.596, 75.028] to (28.64, 27.34, -9.5) mm, rotated rx 180 ry 0 rz 90 deg; joints [74.954, -16.99, 82.839, 0, 24.151, 74.954]
  MoveL 6322 to (28.69, 19.79, -9.5) mm, rotated rx -180 ry 0 rz 90 deg; joints [74.713, -16.949, 82.687, 0, 24.263, 74.713]
  MoveL 6323 to (28.69, 19.79, -6.5) mm, rotated rx -180 ry 0 rz 90 deg; joints [74.713, -17.102, 82.789, 0, 24.313, 74.713]
  Establecer velocidad (1000.0 mm/s)
  MoveL 6324 to (28.69, 19.79, 10) mm, rotated rx 180 ry 0 rz 90 deg; joints [74.713, -17.94, 83.342, 0, 24.598, 74.713]
  Establecer velocidad (66.7 mm/s)
  MoveL 6325 to (11.1, 65.65, 10) mm, rotated rx -180 ry 0 rz 90 deg; joints [76.05, -18.506, 85.465, 0, 23.041, 76.05]
  MoveL 6326 to (11.1, 65.65, -6.25) mm, rotated rx -180 ry 0 rz 90 deg; joints [76.05, -17.674, 84.922, 0, 22.752, 76.05]
  MoveL 6327 to (11.05, 64.13, -6.66) mm, rotated rx -180 ry 0 rz 90 deg; joints [76, -17.647, 84.884, 0, 22.763, 76]
  MoveL 6328 to (11.37, 62.64, -7.06) mm, rotated rx -180 ry 0 rz 90 deg; joints [75.954, -17.614, 84.821, 0, 22.792, 75.954]
  MoveL 6329 to (12.02, 61.27, -7.47) mm, rotated rx 180 ry 0 rz 90 deg; joints [75.915, -17.575, 84.737, 0, 22.838, 75.915]
  MoveL 6330 to (12.95, 60.07, -7.87) mm, rotated rx -180 ry 0 rz 90 deg; joints [75.883, -17.531, 84.635, 0, 22.896, 75.883]
  MoveL 6331 to (14.12, 59.1, -8.28) mm, rotated rx -180 ry 0 rz 90 deg; joints [75.861, -17.484, 84.52, 0, 22.964, 75.861]
  MoveL 6332 to (15.48, 58.42, -8.69) mm, rotated rx 180 ry 0 rz 90 deg; joints [75.85, -17.435, 84.397, 0, 23.038, 75.85]
  MoveL 6333 to (16.96, 58.06, -9.09) mm, rotated rx -180 ry 0 rz 90 deg; joints [75.85, -17.385, 84.271, 0, 23.114, 75.85]
  MoveL 6334 to (18.47, 58.06, -9.5) mm, rotated rx -180 ry 0 rz 90 deg; joints [75.863, -17.336, 84.148, 0, 23.188, 75.863]
  MoveC 6335 to (26.68, 58.86, -9.5) mm, rotated rx 180 ry 0 rz 90 deg; joints [75.956, -17.185, 83.572, 0, 23.613, 75.956] to (34.89, 59.73, -9.5) mm, rotated rx 180 ry 0 rz 90 deg; joints [76.05, -17.032, 82.993, 0, 24.038, 76.05]
  MoveC 6336 to (48.75, 61.5, -9.5) mm, rotated rx -180 ry 0 rz 90 deg; joints [76.218, -16.766, 82.012, 0, 24.755, 76.218] to (62.53, 63.75, -9.5) mm, rotated rx -180 ry 0 rz 90 deg; joints [76.397, -16.496, 81.032, 0, 25.464, 76.397]
  MoveL 6337 to (62.53, 69.41, -9.5) mm, rotated rx -180 ry 0 rz 90 deg; joints [76.578, -16.524, 81.133, 0, 25.391, 76.578]
  MoveC 6338 to (42.89, 70.88, -9.5) mm, rotated rx -180 ry 0 rz 90 deg; joints [76.474, -16.928, 82.608, 0, 24.32, 76.474] to (23.22, 71.73, -9.5) mm, rotated rx 180 ry 0 rz 90 deg; joints [76.347, -17.311, 84.051, 0, 23.26, 76.347]
  MoveC 6339 to (1.14, 72.31, -9.5) mm, rotated rx 180 ry 0 rz 90 deg; joints [76.189, -17.716, 85.635, 0, 22.081, 76.189] to (-20.94, 72.74, -9.5) mm, rotated rx -180 ry 0 rz 90 deg; joints [76.021, -18.097, 87.19, 0, 20.907, 76.021]
  MoveC 6340 to (-23.29, 69.79, -9.5) mm, rotated rx -180 ry 0 rz 90 deg; joints [75.903, -18.124, 87.301, 0, 20.822, 75.903] to (-22.96, 66.04, -9.5) mm, rotated rx -180 ry 0 rz 90 deg; joints [75.781, -18.103, 87.213, 0, 20.89, 75.781]
  MoveL 6341 to (-7.91, 56.39, -9.5) mm, rotated rx -180 ry 0 rz 90 deg; joints [75.588, -17.805, 85.991, 0, 21.814, 75.588]
  MoveL 6342 to (-7.21, 56.02, -9.5) mm, rotated rx -180 ry 0 rz 90 deg; joints [75.581, -17.791, 85.934, 0, 21.856, 75.581]
  MoveL 6343 to (-7.11, 55.99, -9.5) mm, rotated rx 180 ry 0 rz 90 deg; joints [75.581, -17.789, 85.927, 0, 21.862, 75.581]
  MoveC 6344 to (-4.26, 56.18, -9.5) mm, rotated rx 180 ry 0 rz 90 deg; joints [75.612, -17.74, 85.73, 0, 22.009, 75.612] to (-1.42, 56.41, -9.5) mm, rotated rx 180 ry 0 rz 90 deg; joints [75.643, -17.691, 85.534, 0, 22.156, 75.643]
  MoveC 6345 to (8.53, 57.18, -9.5) mm, rotated rx 180 ry 0 rz 90 deg; joints [75.752, -17.515, 84.843, 0, 22.672, 75.752] to (18.47, 58.06, -9.5) mm, rotated rx -180 ry 0 rz 90 deg; joints [75.863, -17.336, 84.148, 0, 23.188, 75.863]
  MoveL 6346 to (17.77, 65.58, -9.5) mm, rotated rx -180 ry 0 rz 90 deg; joints [76.102, -17.384, 84.333, 0, 23.051, 76.102]
  MoveL 6347 to (6.87, 64.62, -9.5) mm, rotated rx 180 ry 0 rz 90 deg; joints [75.982, -17.579, 85.094, 0, 22.485, 75.982]
  MoveL 6348 to (6.87, 64.62, -6.5) mm, rotated rx 180 ry 0 rz 90 deg; joints [75.982, -17.733, 85.196, 0, 22.538, 75.982]
  Establecer velocidad (1000.0 mm/s)
  MoveL 6349 to (6.87, 64.62, 10) mm, rotated rx 180 ry 0 rz 90 deg; joints [75.982, -18.579, 85.747, 0, 22.832, 75.982]
  Establecer velocidad (66.7 mm/s)
  MoveL 6350 to (10, 65.7, 10) mm, rotated rx 180 ry 0 rz 90 deg; joints [76.043, -18.527, 85.544, 0, 22.983, 76.043]
  MoveL 6351 to (10, 65.7, -6.5) mm, rotated rx 180 ry 0 rz 90 deg; joints [76.043, -17.681, 84.992, 0, 22.689, 76.043]
  MoveL 6352 to (9.96, 64.18, -6.91) mm, rotated rx -180 ry 0 rz 90 deg; joints [75.993, -17.654, 84.955, 0, 22.7, 75.993]
  MoveL 6353 to (10.28, 62.7, -7.31) mm, rotated rx 180 ry 0 rz 90 deg; joints [75.947, -17.621, 84.891, 0, 22.729, 75.947]
  MoveL 6354 to (10.93, 61.32, -7.72) mm, rotated rx 180 ry 0 rz 90 deg; joints [75.907, -17.582, 84.807, 0, 22.775, 75.907]
  MoveL 6355 to (11.86, 60.12, -8.13) mm, rotated rx 180 ry 0 rz 90 deg; joints [75.876, -17.539, 84.705, 0, 22.833, 75.876]
  MoveL 6356 to (13.04, 59.16, -8.53) mm, rotated rx 180 ry 0 rz 90 deg; joints [75.854, -17.492, 84.59, 0, 22.902, 75.854]
  MoveL 6357 to (14.4, 58.48, -8.94) mm, rotated rx -180 ry 0 rz 90 deg; joints [75.843, -17.443, 84.467, 0, 22.976, 75.843]
  MoveL 6358 to (15.88, 58.12, -9.34) mm, rotated rx 180 ry 0 rz 90 deg; joints [75.843, -17.393, 84.341, 0, 23.052, 75.843]
  MoveL 6359 to (17.39, 58.13, -9.75) mm, rotated rx 180 ry 0 rz 90 deg; joints [75.856, -17.344, 84.219, 0, 23.125, 75.856]
  MoveL 6360 to (18.46, 58.23, -9.75) mm, rotated rx 180 ry 0 rz 90 deg; joints [75.868, -17.324, 84.144, 0, 23.18, 75.868]
  MoveC 6361 to (27, 59.09, -9.75) mm, rotated rx 180 ry 0 rz 90 deg; joints [75.966, -17.167, 83.545, 0, 23.623, 75.966] to (35.54, 60.02, -9.75) mm, rotated rx -180 ry 0 rz 90 deg; joints [76.065, -17.008, 82.943, 0, 24.065, 76.065]
  MoveC 6362 to (47.63, 61.61, -9.75) mm, rotated rx -180 ry 0 rz 90 deg; joints [76.212, -16.776, 82.087, 0, 24.69, 76.212] to (59.68, 63.56, -9.75) mm, rotated rx 180 ry 0 rz 90 deg; joints [76.369, -16.541, 81.233, 0, 25.309, 76.369]
  MoveL 6363 to (59.68, 69.36, -9.75) mm, rotated rx -180 ry 0 rz 90 deg; joints [76.554, -16.57, 81.336, 0, 25.234, 76.554]
  MoveC 6364 to (41.46, 70.69, -9.75) mm, rotated rx 180 ry 0 rz 90 deg; joints [76.456, -16.943, 82.701, 0, 24.242, 76.456] to (23.22, 71.5, -9.75) mm, rotated rx 180 ry 0 rz 90 deg; joints [76.34, -17.297, 84.038, 0, 23.259, 76.34]
  MoveC 6365 to (1.47, 72.09, -9.75) mm, rotated rx 180 ry 0 rz 90 deg; joints [76.184, -17.696, 85.599, 0, 22.097, 76.184] to (-20.27, 72.55, -9.75) mm, rotated rx 180 ry 0 rz 90 deg; joints [76.021, -18.072, 87.131, 0, 20.941, 76.021]
  MoveC 6366 to (-22.64, 69.64, -9.75) mm, rotated rx -180 ry 0 rz 90 deg; joints [75.904, -18.099, 87.245, 0, 20.854, 75.904] to (-22.32, 65.91, -9.75) mm, rotated rx -180 ry 0 rz 90 deg; joints [75.782, -18.078, 87.158, 0, 20.921, 75.782]
  MoveL 6367 to (-7.48, 56.39, -9.75) mm, rotated rx -180 ry 0 rz 90 deg; joints [75.591, -17.784, 85.952, 0, 21.832, 75.591]
  MoveL 6368 to (-6.95, 56.13, -9.75) mm, rotated rx -180 ry 0 rz 90 deg; joints [75.587, -17.774, 85.91, 0, 21.864, 75.587]
  MoveC 6369 to (5.76, 57.1, -9.75) mm, rotated rx 180 ry 0 rz 90 deg; joints [75.726, -17.552, 85.03, 0, 22.523, 75.726] to (18.46, 58.23, -9.75) mm, rotated rx 180 ry 0 rz 90 deg; joints [75.868, -17.324, 84.144, 0, 23.18, 75.868]
  MoveL 6370 to (17.74, 65.75, -9.75) mm, rotated rx -180 ry 0 rz 90 deg; joints [76.108, -17.373, 84.33, 0, 23.043, 76.108]
  MoveL 6371 to (3.47, 64.49, -9.75) mm, rotated rx -180 ry 0 rz 90 deg; joints [75.95, -17.627, 85.324, 0, 22.303, 75.95]
  MoveL 6372 to (3.47, 64.49, -6.75) mm, rotated rx 180 ry 0 rz 90 deg; joints [75.95, -17.781, 85.426, 0, 22.355, 75.95]
  Establecer velocidad (1000.0 mm/s)
  MoveL 6373 to (3.47, 64.49, 10) mm, rotated rx -180 ry 0 rz 90 deg; joints [75.95, -18.641, 85.986, 0, 22.655, 75.95]
  Establecer velocidad (66.7 mm/s)
  MoveL 6374 to (35.58, 18.9, 10) mm, rotated rx -180 ry 0 rz 90 deg; joints [74.744, -17.798, 82.824, 0, 24.974, 74.744]
  MoveL 6375 to (35.58, 18.9, -6.5) mm, rotated rx 180 ry 0 rz 90 deg; joints [74.744, -16.961, 82.271, 0, 24.691, 74.744]
  MoveL 6376 to (35.75, 20.41, -6.91) mm, rotated rx -180 ry 0 rz 90 deg; joints [74.794, -16.945, 82.274, 0, 24.671, 74.794]
  MoveL 6377 to (35.56, 21.92, -7.31) mm, rotated rx -180 ry 0 rz 90 deg; joints [74.84, -16.937, 82.304, 0, 24.633, 74.84]
  MoveL 6378 to (35.04, 23.34, -7.72) mm, rotated rx 180 ry 0 rz 90 deg; joints [74.881, -16.934, 82.356, 0, 24.578, 74.881]
  MoveL 6379 to (34.22, 24.62, -8.13) mm, rotated rx -180 ry 0 rz 90 deg; joints [74.915, -16.937, 82.427, 0, 24.509, 74.915]
  MoveL 6380 to (33.13, 25.68, -8.53) mm, rotated rx -180 ry 0 rz 90 deg; joints [74.94, -16.943, 82.513, 0, 24.43, 74.94]
  MoveL 6381 to (31.84, 26.48, -8.94) mm, rotated rx -180 ry 0 rz 90 deg; joints [74.954, -16.952, 82.609, 0, 24.343, 74.954]
  MoveL 6382 to (30.4, 26.97, -9.34) mm, rotated rx -180 ry 0 rz 90 deg; joints [74.958, -16.962, 82.709, 0, 24.253, 74.958]
  MoveL 6383 to (28.89, 27.1, -9.75) mm, rotated rx 180 ry 0 rz 90 deg; joints [74.949, -16.971, 82.808, 0, 24.164, 74.949]
  MoveC 6384 to (20.84, 27.04, -9.75) mm, rotated rx 180 ry 0 rz 90 deg; joints [74.877, -17.126, 83.388, 0, 23.738, 74.877] to (12.79, 26.94, -9.75) mm, rotated rx 180 ry 0 rz 90 deg; joints [74.803, -17.277, 83.963, 0, 23.314, 74.803]
  MoveC 6385 to (10.12, 25.62, -9.75) mm, rotated rx 180 ry 0 rz 90 deg; joints [74.737, -17.321, 84.129, 0, 23.192, 74.737] to (9.33, 22.74, -9.75) mm, rotated rx -180 ry 0 rz 90 deg; joints [74.637, -17.321, 84.129, 0, 23.192, 74.637]
  MoveL 6386 to (9.49, 22.27, -9.75) mm, rotated rx -180 ry 0 rz 90 deg; joints [74.623, -17.315, 84.108, 0, 23.207, 74.623]
  MoveL 6387 to (13.31, 11.85, -9.75) mm, rotated rx 180 ry 0 rz 90 deg; joints [74.32, -17.189, 83.628, 0, 23.562, 74.32]
  MoveL 6388 to (13.7, 10.8, -9.75) mm, rotated rx 180 ry 0 rz 90 deg; joints [74.29, -17.177, 83.579, 0, 23.598, 74.29]
  MoveC 6389 to (14.2, 9.89, -9.75) mm, rotated rx -180 ry 0 rz 90 deg; joints [74.265, -17.162, 83.525, 0, 23.637, 74.265] to (14.93, 9.15, -9.75) mm, rotated rx 180 ry 0 rz 90 deg; joints [74.248, -17.144, 83.457, 0, 23.687, 74.248]
  MoveL 6390 to (28.4, -0.99, -9.75) mm, rotated rx -180 ry 0 rz 90 deg; joints [74.046, -16.828, 82.278, 0, 24.551, 74.046]
  MoveC 6391 to (28.92, -1.29, -9.75) mm, rotated rx 180 ry 0 rz 90 deg; joints [74.041, -16.817, 82.234, 0, 24.582, 74.041] to (29.48, -1.45, -9.75) mm, rotated rx -180 ry 0 rz 90 deg; joints [74.041, -16.804, 82.189, 0, 24.615, 74.041]
  MoveC 6392 to (31.76, -1.19, -9.75) mm, rotated rx -180 ry 0 rz 90 deg; joints [74.07, -16.761, 82.029, 0, 24.731, 74.07] to (33.54, 0.25, -9.75) mm, rotated rx 180 ry 0 rz 90 deg; joints [74.132, -16.734, 81.93, 0, 24.804, 74.132]
  MoveL 6393 to (44.88, 16.58, -9.75) mm, rotated rx -180 ry 0 rz 90 deg; joints [74.751, -16.597, 81.432, 0, 25.165, 74.751]
  MoveL 6394 to (47.46, 20.32, -9.75) mm, rotated rx -180 ry 0 rz 90 deg; joints [74.892, -16.565, 81.317, 0, 25.248, 74.892]
  MoveC 6395 to (47.85, 21.18, -9.75) mm, rotated rx 180 ry 0 rz 90 deg; joints [74.923, -16.562, 81.306, 0, 25.256, 74.923] to (47.9, 22.13, -9.75) mm, rotated rx 180 ry 0 rz 90 deg; joints [74.953, -16.566, 81.32, 0, 25.245, 74.953]
  MoveL 6396 to (47.8, 22.91, -9.75) mm, rotated rx 180 ry 0 rz 90 deg; joints [74.977, -16.572, 81.343, 0, 25.229, 74.977]
  MoveC 6397 to (46.89, 25.35, -9.75) mm, rotated rx 180 ry 0 rz 90 deg; joints [75.047, -16.604, 81.458, 0, 25.146, 75.047] to (44.98, 27.13, -9.75) mm, rotated rx 180 ry 0 rz 90 deg; joints [75.087, -16.652, 81.633, 0, 25.019, 75.087]
  MoveC 6398 to (36.94, 27.13, -9.75) mm, rotated rx 180 ry 0 rz 90 deg; joints [75.019, -16.813, 82.223, 0, 24.591, 75.019] to (28.89, 27.1, -9.75) mm, rotated rx 180 ry 0 rz 90 deg; joints [74.949, -16.971, 82.808, 0, 24.164, 74.949]
  MoveL 6399 to (28.93, 19.55, -9.75) mm, rotated rx 180 ry 0 rz 90 deg; joints [74.707, -16.931, 82.656, 0, 24.275, 74.707]
  MoveL 6400 to (28.93, 19.55, -6.75) mm, rotated rx 180 ry 0 rz 90 deg; joints [74.707, -17.083, 82.758, 0, 24.325, 74.707]
  Establecer velocidad (1000.0 mm/s)
  MoveL 6401 to (28.93, 19.55, 10) mm, rotated rx -180 ry 0 rz 90 deg; joints [74.707, -17.934, 83.32, 0, 24.614, 74.707]
  Establecer velocidad (66.7 mm/s)
  MoveL 6402 to (59.68, -25.57, 10) mm, rotated rx -180 ry 0 rz 90 deg; joints [73.558, -17.029, 80.115, 0, 26.914, 73.558]
  MoveL 6403 to (59.68, -25.57, -6.5) mm, rotated rx 180 ry 0 rz 90 deg; joints [73.558, -16.2, 79.559, 0, 26.642, 73.558]
  MoveL 6404 to (59.68, -25.57, -9.75) mm, rotated rx -180 ry 0 rz 90 deg; joints [73.558, -16.037, 79.447, 0, 26.589, 73.558]
  MoveL 6405 to (59.68, -21.58, -9.75) mm, rotated rx -180 ry 0 rz 90 deg; joints [73.682, -16.062, 79.535, 0, 26.527, 73.682]
  MoveL 6406 to (57.84, -24.04, -9.75) mm, rotated rx -180 ry 0 rz 90 deg; joints [73.589, -16.086, 79.619, 0, 26.467, 73.589]
  MoveC 6407 to (57.27, -25.68, -9.75) mm, rotated rx 180 ry 0 rz 90 deg; joints [73.533, -16.088, 79.625, 0, 26.463, 73.533] to (57.77, -27.35, -9.75) mm, rotated rx 180 ry 0 rz 90 deg; joints [73.485, -16.066, 79.55, 0, 26.516, 73.485]
  MoveL 6408 to (58.19, -27.96, -9.75) mm, rotated rx 180 ry 0 rz 90 deg; joints [73.47, -16.053, 79.505, 0, 26.548, 73.47]
  MoveL 6409 to (58.28, -28.05, -9.75) mm, rotated rx -180 ry 0 rz 90 deg; joints [73.468, -16.051, 79.497, 0, 26.554, 73.468]
  MoveL 6410 to (59.68, -29.57, -9.75) mm, rotated rx 180 ry 0 rz 90 deg; joints [73.434, -16.011, 79.359, 0, 26.653, 73.434]
  MoveL 6411 to (59.68, -25.57, -9.75) mm, rotated rx -180 ry 0 rz 90 deg; joints [73.558, -16.037, 79.447, 0, 26.589, 73.558]
  MoveL 6412 to (59.68, -25.57, -6.75) mm, rotated rx -180 ry 0 rz 90 deg; joints [73.558, -16.188, 79.55, 0, 26.638, 73.558]
  Establecer velocidad (1000.0 mm/s)
  MoveL 6413 to (59.68, -25.57, 10) mm, rotated rx -180 ry 0 rz 90 deg; joints [73.558, -17.029, 80.115, 0, 26.914, 73.558]
  Establecer velocidad (66.7 mm/s)
  MoveL 6414 to (15.39, -63.74, 10) mm, rotated rx -180 ry 0 rz 90 deg; joints [71.935, -17.706, 82.494, 0, 25.212, 71.935]
  MoveL 6415 to (15.39, -63.74, -6.5) mm, rotated rx 180 ry 0 rz 90 deg; joints [71.935, -16.871, 81.941, 0, 24.93, 71.935]
  MoveL 6416 to (15.25, -65.26, -6.91) mm, rotated rx -180 ry 0 rz 90 deg; joints [71.887, -16.843, 81.901, 0, 24.942, 71.887]
  MoveL 6417 to (15.48, -66.76, -7.31) mm, rotated rx 180 ry 0 rz 90 deg; joints [71.842, -16.809, 81.835, 0, 24.973, 71.842]
  MoveL 6418 to (16.04, -68.17, -7.72) mm, rotated rx 180 ry 0 rz 90 deg; joints [71.803, -16.768, 81.748, 0, 25.02, 71.803]
  MoveL 6419 to (16.89, -69.43, -8.13) mm, rotated rx 180 ry 0 rz 90 deg; joints [71.773, -16.722, 81.643, 0, 25.079, 71.773]
  MoveL 6420 to (18, -70.46, -8.53) mm, rotated rx -180 ry 0 rz 90 deg; joints [71.752, -16.672, 81.524, 0, 25.148, 71.752]
  MoveL 6421 to (19.31, -71.23, -8.94) mm, rotated rx 180 ry 0 rz 90 deg; joints [71.741, -16.62, 81.397, 0, 25.224, 71.741]
  MoveL 6422 to (20.76, -71.69, -9.34) mm, rotated rx 180 ry 0 rz 90 deg; joints [71.742, -16.568, 81.267, 0, 25.301, 71.742]
  MoveL 6423 to (22.28, -71.78, -9.75) mm, rotated rx -180 ry 0 rz 90 deg; joints [71.755, -16.516, 81.141, 0, 25.375, 71.755]
  MoveC 6424 to (32.84, -71.43, -9.75) mm, rotated rx 180 ry 0 rz 90 deg; joints [71.873, -16.302, 80.378, 0, 25.924, 71.873] to (43.4, -71.03, -9.75) mm, rotated rx 180 ry 0 rz 90 deg; joints [71.993, -16.083, 79.61, 0, 26.474, 71.993]
  MoveC 6425 to (45.72, -68.09, -9.75) mm, rotated rx -180 ry 0 rz 90 deg; joints [72.107, -16.054, 79.508, 0, 26.546, 72.107] to (45.86, -64.34, -9.75) mm, rotated rx 180 ry 0 rz 90 deg; joints [72.224, -16.077, 79.588, 0, 26.49, 72.224]
  MoveC 6426 to (35.12, -51.34, -9.75) mm, rotated rx -180 ry 0 rz 90 deg; joints [72.522, -16.388, 80.684, 0, 25.704, 72.522] to (24.28, -38.43, -9.75) mm, rotated rx 180 ry 0 rz 90 deg; joints [72.821, -16.689, 81.768, 0, 24.921, 72.821]
  MoveC 6427 to (23.91, -38.03, -9.75) mm, rotated rx -180 ry 0 rz 90 deg; joints [72.83, -16.699, 81.804, 0, 24.895, 72.83] to (23.51, -37.66, -9.75) mm, rotated rx 180 ry 0 rz 90 deg; joints [72.837, -16.709, 81.842, 0, 24.868, 72.837]
  MoveL 6428 to (13.14, -29.22, -9.75) mm, rotated rx 180 ry 0 rz 90 deg; joints [73.004, -16.963, 82.777, 0, 24.186, 73.004]
  MoveC 6429 to (10.44, -28.73, -9.75) mm, rotated rx 180 ry 0 rz 90 deg; joints [72.993, -17.018, 82.981, 0, 24.037, 72.993] to (8.05, -30.07, -9.75) mm, rotated rx 180 ry 0 rz 90 deg; joints [72.927, -17.056, 83.123, 0, 23.933, 72.927]
  MoveC 6430 to (7.8, -30.56, -9.75) mm, rotated rx -180 ry 0 rz 90 deg; joints [72.909, -17.058, 83.13, 0, 23.928, 72.909] to (7.62, -31.08, -9.75) mm, rotated rx -180 ry 0 rz 90 deg; joints [72.891, -17.058, 83.131, 0, 23.927, 72.891]
  MoveL 6431 to (5.92, -37.43, -9.75) mm, rotated rx 180 ry 0 rz 90 deg; joints [72.672, -17.053, 83.113, 0, 23.94, 72.672]
  MoveL 6432 to (-2.34, -68.04, -9.75) mm, rotated rx -180 ry 0 rz 90 deg; joints [71.616, -17.022, 82.998, 0, 24.024, 71.616]
  MoveC 6433 to (-2.33, -69.76, -9.75) mm, rotated rx 180 ry 0 rz 90 deg; joints [71.562, -17.011, 82.957, 0, 24.055, 71.562] to (-1.42, -71.22, -9.75) mm, rotated rx -180 ry 0 rz 90 deg; joints [71.526, -16.985, 82.858, 0, 24.127, 71.526]
  MoveC 6434 to (-0.26, -72.04, -9.75) mm, rotated rx 180 ry 0 rz 90 deg; joints [71.512, -16.957, 82.755, 0, 24.202, 71.512] to (1.14, -72.31, -9.75) mm, rotated rx 180 ry 0 rz 90 deg; joints [71.518, -16.929, 82.649, 0, 24.28, 71.518]
  MoveC 6435 to (11.71, -72.07, -9.75) mm, rotated rx 180 ry 0 rz 90 deg; joints [71.636, -16.725, 81.898, 0, 24.827, 71.636] to (22.28, -71.78, -9.75) mm, rotated rx -180 ry 0 rz 90 deg; joints [71.755, -16.516, 81.141, 0, 25.375, 71.755]
  MoveL 6436 to (22.05, -64.23, -9.75) mm, rotated rx 180 ry 0 rz 90 deg; joints [71.988, -16.57, 81.337, 0, 25.234, 71.988]
  MoveL 6437 to (22.05, -64.23, -6.75) mm, rotated rx -180 ry 0 rz 90 deg; joints [71.988, -16.722, 81.439, 0, 25.283, 71.988]
  Establecer velocidad (1000.0 mm/s)
  MoveL 6438 to (22.05, -64.23, 10) mm, rotated rx 180 ry 0 rz 90 deg; joints [71.988, -17.569, 82.001, 0, 25.567, 71.988]
  Establecer velocidad (66.7 mm/s)
  MoveL 6439 to (-36.73, -51.61, 10) mm, rotated rx -180 ry 0 rz 90 deg; joints [71.778, -18.759, 86.449, 0, 22.31, 71.778]
  MoveL 6440 to (-36.73, -51.61, -6.5) mm, rotated rx -180 ry 0 rz 90 deg; joints [71.778, -17.91, 85.898, 0, 22.013, 71.778]
  MoveL 6441 to (-35.32, -52.16, -6.91) mm, rotated rx -180 ry 0 rz 90 deg; joints [71.775, -17.862, 85.774, 0, 22.088, 71.775]
  MoveL 6442 to (-33.81, -52.36, -7.31) mm, rotated rx -180 ry 0 rz 90 deg; joints [71.785, -17.814, 85.651, 0, 22.162, 71.785]
  MoveL 6443 to (-32.3, -52.23, -7.72) mm, rotated rx 180 ry 0 rz 90 deg; joints [71.805, -17.767, 85.536, 0, 22.231, 71.805]
  MoveL 6444 to (-30.85, -51.76, -8.13) mm, rotated rx 180 ry 0 rz 90 deg; joints [71.835, -17.724, 85.432, 0, 22.291, 71.835]
  MoveL 6445 to (-29.55, -50.99, -8.53) mm, rotated rx 180 ry 0 rz 90 deg; joints [71.874, -17.684, 85.346, 0, 22.339, 71.874]
  MoveL 6446 to (-28.44, -49.94, -8.94) mm, rotated rx -180 ry 0 rz 90 deg; joints [71.92, -17.65, 85.279, 0, 22.371, 71.92]
  MoveL 6447 to (-27.6, -48.68, -9.34) mm, rotated rx -180 ry 0 rz 90 deg; joints [71.969, -17.622, 85.235, 0, 22.387, 71.969]
  MoveL 6448 to (-27.08, -47.25, -9.75) mm, rotated rx -180 ry 0 rz 90 deg; joints [72.021, -17.6, 85.218, 0, 22.382, 72.021]
  MoveL 6449 to (-26.26, -44.07, -9.75) mm, rotated rx 180 ry 0 rz 90 deg; joints [72.132, -17.604, 85.232, 0, 22.372, 72.132]
  MoveL 6450 to (-25.11, -39.61, -9.75) mm, rotated rx -180 ry 0 rz 90 deg; joints [72.287, -17.609, 85.252, 0, 22.357, 72.287]
  MoveL 6451 to (-21.22, -24.64, -9.75) mm, rotated rx 180 ry 0 rz 90 deg; joints [72.812, -17.623, 85.308, 0, 22.315, 72.812]
  MoveL 6452 to (-21.15, -24.17, -9.75) mm, rotated rx 180 ry 0 rz 90 deg; joints [72.828, -17.624, 85.313, 0, 22.311, 72.828]
  MoveC 6453 to (-22.2, -21.68, -9.75) mm, rotated rx -180 ry 0 rz 90 deg; joints [72.898, -17.656, 85.441, 0, 22.216, 72.898] to (-24.64, -20.5, -9.75) mm, rotated rx 180 ry 0 rz 90 deg; joints [72.912, -17.705, 85.635, 0, 22.07, 72.912]
  MoveL 6454 to (-26.06, -20.76, -9.75) mm, rotated rx 180 ry 0 rz 90 deg; joints [72.889, -17.728, 85.729, 0, 22, 72.889]
  MoveL 6455 to (-33.33, -22.27, -9.75) mm, rotated rx -180 ry 0 rz 90 deg; joints [72.767, -17.845, 86.2, 0, 21.645, 72.767]
  MoveL 6456 to (-71.02, -30.17, -9.75) mm, rotated rx 180 ry 0 rz 90 deg; joints [72.114, -18.416, 88.596, 0, 19.82, 72.114]
  MoveC 6457 to (-72.8, -31.25, -9.75) mm, rotated rx 180 ry 0 rz 90 deg; joints [72.059, -18.438, 88.692, 0, 19.746, 72.059] to (-73.49, -33.21, -9.75) mm, rotated rx -180 ry 0 rz 90 deg; joints [71.987, -18.439, 88.696, 0, 19.743, 71.987]
  MoveL 6458 to (-73.49, -69.82, -9.75) mm, rotated rx -180 ry 0 rz 90 deg; joints [70.78, -18.247, 87.869, 0, 20.378, 70.78]
  MoveC 6459 to (-72.56, -72.06, -9.75) mm, rotated rx 180 ry 0 rz 90 deg; joints [70.717, -18.22, 87.754, 0, 20.466, 70.717] to (-70.31, -72.97, -9.75) mm, rotated rx -180 ry 0 rz 90 deg; joints [70.713, -18.179, 87.581, 0, 20.598, 70.713]
  MoveL 6460 to (-37.43, -72.62, -9.75) mm, rotated rx 180 ry 0 rz 90 deg; joints [71.093, -17.633, 85.349, 0, 22.284, 71.093]
  MoveL 6461 to (-36.05, -72.59, -9.75) mm, rotated rx 180 ry 0 rz 90 deg; joints [71.109, -17.609, 85.253, 0, 22.356, 71.109]
  MoveC 6462 to (-34.19, -71.95, -9.75) mm, rotated rx 180 ry 0 rz 90 deg; joints [71.15, -17.58, 85.14, 0, 22.44, 71.15] to (-33.09, -70.32, -9.75) mm, rotated rx 180 ry 0 rz 90 deg; joints [71.214, -17.571, 85.103, 0, 22.468, 71.214]
  MoveL 6463 to (-32.9, -69.65, -9.75) mm, rotated rx 180 ry 0 rz 90 deg; joints [71.238, -17.571, 85.105, 0, 22.466, 71.238]
  MoveL 6464 to (-27.08, -47.25, -9.75) mm, rotated rx -180 ry 0 rz 90 deg; joints [72.021, -17.6, 85.218, 0, 22.382, 72.021]
  MoveL 6465 to (-34.39, -45.35, -9.75) mm, rotated rx -180 ry 0 rz 90 deg; joints [72.005, -17.738, 85.767, 0, 21.971, 72.005]
  MoveL 6466 to (-34.39, -45.35, -6.75) mm, rotated rx 180 ry 0 rz 90 deg; joints [72.005, -17.893, 85.869, 0, 22.024, 72.005]
  Establecer velocidad (1000.0 mm/s)
  MoveL 6467 to (-34.39, -45.35, 10) mm, rotated rx -180 ry 0 rz 90 deg; joints [72.005, -18.754, 86.429, 0, 22.325, 72.005]
  Establecer velocidad (66.7 mm/s)
  MoveL 6468 to (-65.26, 35.78, 10) mm, rotated rx 180 ry 0 rz 90 deg; joints [74.384, -19.663, 90.204, 0, 19.459, 74.384]
  MoveL 6469 to (-65.26, 35.78, -6.5) mm, rotated rx 180 ry 0 rz 90 deg; joints [74.384, -18.8, 89.652, 0, 19.148, 74.384]
  MoveL 6470 to (-66.76, 35.97, -6.91) mm, rotated rx 180 ry 0 rz 90 deg; joints [74.376, -18.802, 89.743, 0, 19.059, 74.376]
  MoveL 6471 to (-68.27, 35.78, -7.31) mm, rotated rx -180 ry 0 rz 90 deg; joints [74.355, -18.802, 89.827, 0, 18.975, 74.355]
  MoveL 6472 to (-69.7, 35.27, -7.72) mm, rotated rx 180 ry 0 rz 90 deg; joints [74.324, -18.8, 89.9, 0, 18.9, 74.324]
  MoveL 6473 to (-70.98, 34.46, -8.13) mm, rotated rx 180 ry 0 rz 90 deg; joints [74.284, -18.794, 89.956, 0, 18.838, 74.284]
  MoveL 6474 to (-72.05, 33.38, -8.53) mm, rotated rx -180 ry 0 rz 90 deg; joints [74.238, -18.784, 89.994, 0, 18.79, 74.238]
  MoveL 6475 to (-72.86, 32.09, -8.94) mm, rotated rx -180 ry 0 rz 90 deg; joints [74.186, -18.769, 90.01, 0, 18.76, 74.186]
  MoveL 6476 to (-73.36, 30.65, -9.34) mm, rotated rx 180 ry 0 rz 90 deg; joints [74.132, -18.749, 90.002, 0, 18.748, 74.132]
  MoveL 6477 to (-73.49, 29.14, -9.75) mm, rotated rx 180 ry 0 rz 90 deg; joints [74.08, -18.724, 89.968, 0, 18.755, 74.08]
  MoveL 6478 to (-73.49, 2.37, -9.75) mm, rotated rx 180 ry 0 rz 90 deg; joints [73.175, -18.608, 89.443, 0, 19.165, 73.175]
  MoveL 6479 to (-73.46, 1.42, -9.75) mm, rotated rx 180 ry 0 rz 90 deg; joints [73.144, -18.603, 89.421, 0, 19.182, 73.144]
  MoveC 6480 to (-72.25, -0.46, -9.75) mm, rotated rx -180 ry 0 rz 90 deg; joints [73.093, -18.576, 89.302, 0, 19.274, 73.093] to (-70.13, -1.17, -9.75) mm, rotated rx 180 ry 0 rz 90 deg; joints [73.091, -18.541, 89.145, 0, 19.396, 73.091]
  MoveL 6481 to (-69.65, -1.07, -9.75) mm, rotated rx -180 ry 0 rz 90 deg; joints [73.099, -18.534, 89.115, 0, 19.419, 73.099]
  MoveL 6482 to (-51.65, 3.09, -9.75) mm, rotated rx -180 ry 0 rz 90 deg; joints [73.419, -18.274, 87.984, 0, 20.29, 73.419]
  MoveL 6483 to (-24.17, 9.53, -9.75) mm, rotated rx -180 ry 0 rz 90 deg; joints [73.898, -17.851, 86.225, 0, 21.627, 73.898]
  MoveL 6484 to (-22.45, 9.95, -9.75) mm, rotated rx 180 ry 0 rz 90 deg; joints [73.928, -17.824, 86.114, 0, 21.71, 73.928]
  MoveC 6485 to (-20.45, 11.73, -9.75) mm, rotated rx 180 ry 0 rz 90 deg; joints [74.005, -17.799, 86.01, 0, 21.788, 74.005] to (-20.37, 14.4, -9.75) mm, rotated rx 180 ry 0 rz 90 deg; joints [74.093, -17.81, 86.058, 0, 21.752, 74.093]
  MoveL 6486 to (-26.39, 31.26, -9.75) mm, rotated rx 180 ry 0 rz 90 deg; joints [74.594, -17.993, 86.804, 0, 21.189, 74.594]
  MoveC 6487 to (-26.71, 31.96, -9.75) mm, rotated rx 180 ry 0 rz 90 deg; joints [74.614, -18.002, 86.84, 0, 21.162, 74.614] to (-27.15, 32.59, -9.75) mm, rotated rx -180 ry 0 rz 90 deg; joints [74.631, -18.012, 86.883, 0, 21.129, 74.631]
  MoveC 6488 to (-27.68, 33.01, -9.75) mm, rotated rx 180 ry 0 rz 90 deg; joints [74.64, -18.023, 86.927, 0, 21.096, 74.64] to (-28.23, 33.39, -9.75) mm, rotated rx 180 ry 0 rz 90 deg; joints [74.647, -18.034, 86.972, 0, 21.062, 74.647]
  MoveL 6489 to (-35.54, 38.13, -9.75) mm, rotated rx 180 ry 0 rz 90 deg; joints [74.738, -18.176, 87.566, 0, 20.61, 74.738]
  MoveL 6490 to (-68.7, 59.48, -9.75) mm, rotated rx 180 ry 0 rz 90 deg; joints [75.158, -18.776, 90.206, 0, 18.569, 75.158]
  MoveL 6491 to (-69.07, 59.7, -9.75) mm, rotated rx 180 ry 0 rz 90 deg; joints [75.163, -18.782, 90.234, 0, 18.547, 75.163]
  MoveC 6492 to (-71.49, 59.46, -9.75) mm, rotated rx 180 ry 0 rz 90 deg; joints [75.132, -18.816, 90.392, 0, 18.424, 75.132] to (-73.27, 57.8, -9.75) mm, rotated rx 180 ry 0 rz 90 deg; joints [75.059, -18.835, 90.482, 0, 18.353, 75.059]
  MoveC 6493 to (-73.45, 57.35, -9.75) mm, rotated rx 180 ry 0 rz 90 deg; joints [75.042, -18.836, 90.486, 0, 18.35, 75.042] to (-73.49, 56.86, -9.75) mm, rotated rx 180 ry 0 rz 90 deg; joints [75.025, -18.835, 90.48, 0, 18.355, 75.025]
  MoveL 6494 to (-73.49, 29.14, -9.75) mm, rotated rx 180 ry 0 rz 90 deg; joints [74.08, -18.724, 89.968, 0, 18.755, 74.08]
  MoveL 6495 to (-65.95, 29.14, -9.75) mm, rotated rx -180 ry 0 rz 90 deg; joints [74.153, -18.612, 89.463, 0, 19.149, 74.153]
  MoveL 6496 to (-65.95, 29.14, -6.75) mm, rotated rx 180 ry 0 rz 90 deg; joints [74.153, -18.769, 89.565, 0, 19.205, 74.153]
  Establecer velocidad (1000.0 mm/s)
  MoveL 6497 to (-65.95, 29.14, 10) mm, rotated rx 180 ry 0 rz 90 deg; joints [74.153, -19.645, 90.125, 0, 19.52, 74.153]
  Establecer velocidad (66.7 mm/s)
  MoveL 6498 to (-65.09, 35.78, 10) mm, rotated rx 180 ry 0 rz 90 deg; joints [74.385, -19.661, 90.193, 0, 19.467, 74.385]
  MoveL 6499 to (-65.09, 35.78, -6.75) mm, rotated rx 180 ry 0 rz 90 deg; joints [74.385, -18.784, 89.633, 0, 19.151, 74.385]
  MoveL 6500 to (-66.6, 35.97, -7.16) mm, rotated rx 180 ry 0 rz 90 deg; joints [74.377, -18.786, 89.724, 0, 19.063, 74.377]
  MoveL 6501 to (-68.11, 35.78, -7.56) mm, rotated rx -180 ry 0 rz 90 deg; joints [74.357, -18.787, 89.808, 0, 18.979, 74.357]
  MoveL 6502 to (-69.54, 35.27, -7.97) mm, rotated rx -180 ry 0 rz 90 deg; joints [74.326, -18.785, 89.88, 0, 18.904, 74.326]
  MoveL 6503 to (-70.82, 34.46, -8.37) mm, rotated rx 180 ry 0 rz 90 deg; joints [74.286, -18.779, 89.937, 0, 18.842, 74.286]
  MoveL 6504 to (-71.89, 33.38, -8.78) mm, rotated rx -180 ry 0 rz 90 deg; joints [74.239, -18.769, 89.974, 0, 18.794, 74.239]
  MoveL 6505 to (-72.69, 32.09, -9.19) mm, rotated rx 180 ry 0 rz 90 deg; joints [74.188, -18.754, 89.99, 0, 18.764, 74.188]
  MoveL 6506 to (-73.19, 30.65, -9.59) mm, rotated rx 180 ry 0 rz 90 deg; joints [74.134, -18.734, 89.982, 0, 18.752, 74.134]
  MoveL 6507 to (-73.33, 29.14, -10) mm, rotated rx 180 ry 0 rz 90 deg; joints [74.082, -18.708, 89.949, 0, 18.759, 74.082]
  MoveL 6508 to (-73.33, 3.32, -10) mm, rotated rx -180 ry 0 rz 90 deg; joints [73.209, -18.596, 89.442, 0, 19.154, 73.209]
  MoveL 6509 to (-73.33, 2.37, -10) mm, rotated rx 180 ry 0 rz 90 deg; joints [73.177, -18.592, 89.423, 0, 19.169, 73.177]
  MoveC 6510 to (-72.44, 0.01, -10) mm, rotated rx 180 ry 0 rz 90 deg; joints [73.107, -18.568, 89.316, 0, 19.252, 73.107] to (-70.13, -1.01, -10) mm, rotated rx 180 ry 0 rz 90 deg; joints [73.096, -18.529, 89.14, 0, 19.389, 73.096]
  MoveL 6511 to (-68.7, -0.72, -10) mm, rotated rx 180 ry 0 rz 90 deg; joints [73.12, -18.508, 89.051, 0, 19.458, 73.12]
  MoveC 6512 to (-45.77, 4.61, -10) mm, rotated rx -180 ry 0 rz 90 deg; joints [73.527, -18.174, 87.606, 0, 20.568, 73.527] to (-22.86, 10.01, -10) mm, rotated rx -180 ry 0 rz 90 deg; joints [73.926, -17.819, 86.135, 0, 21.684, 73.926]
  MoveC 6513 to (-22.34, 10.18, -10) mm, rotated rx -180 ry 0 rz 90 deg; joints [73.936, -17.811, 86.102, 0, 21.708, 73.936] to (-21.86, 10.42, -10) mm, rotated rx 180 ry 0 rz 90 deg; joints [73.949, -17.803, 86.074, 0, 21.73, 73.949]
  MoveC 6514 to (-20.65, 11.88, -10) mm, rotated rx 180 ry 0 rz 90 deg; joints [74.008, -17.79, 86.019, 0, 21.771, 74.008] to (-20.35, 13.74, -10) mm, rotated rx -180 ry 0 rz 90 deg; joints [74.072, -17.794, 86.035, 0, 21.759, 74.072]
  MoveL 6515 to (-20.65, 14.69, -10) mm, rotated rx 180 ry 0 rz 90 deg; joints [74.1, -17.804, 86.074, 0, 21.729, 74.1]
  MoveL 6516 to (-26.54, 31.24, -10) mm, rotated rx 180 ry 0 rz 90 deg; joints [74.592, -17.983, 86.806, 0, 21.177, 74.592]
  MoveC 6517 to (-26.85, 31.89, -10) mm, rotated rx -180 ry 0 rz 90 deg; joints [74.61, -17.991, 86.84, 0, 21.151, 74.61] to (-27.27, 32.48, -10) mm, rotated rx 180 ry 0 rz 90 deg; joints [74.626, -18.001, 86.88, 0, 21.12, 74.626]
  MoveC 6518 to (-27.75, 32.86, -10) mm, rotated rx 180 ry 0 rz 90 deg; joints [74.634, -18.01, 86.92, 0, 21.09, 74.634] to (-28.25, 33.21, -10) mm, rotated rx 180 ry 0 rz 90 deg; joints [74.641, -18.02, 86.962, 0, 21.059, 74.641]
  MoveL 6519 to (-31.83, 35.54, -10) mm, rotated rx 180 ry 0 rz 90 deg; joints [74.686, -18.09, 87.253, 0, 20.837, 74.686]
  MoveL 6520 to (-64.14, 56.39, -10) mm, rotated rx 180 ry 0 rz 90 deg; joints [75.094, -18.684, 89.837, 0, 18.847, 75.094]
  MoveL 6521 to (-68.94, 59.45, -10) mm, rotated rx 180 ry 0 rz 90 deg; joints [75.155, -18.766, 90.213, 0, 18.553, 75.155]
  MoveC 6522 to (-71.28, 59.24, -10) mm, rotated rx -180 ry 0 rz 90 deg; joints [75.127, -18.799, 90.366, 0, 18.433, 75.127] to (-73.05, 57.69, -10) mm, rotated rx 180 ry 0 rz 90 deg; joints [75.058, -18.819, 90.457, 0, 18.362, 75.058]
  MoveC 6523 to (-73.25, 57.22, -10) mm, rotated rx 180 ry 0 rz 90 deg; joints [75.04, -18.82, 90.462, 0, 18.358, 75.04] to (-73.33, 56.71, -10) mm, rotated rx -180 ry 0 rz 90 deg; joints [75.021, -18.819, 90.458, 0, 18.361, 75.021]
  MoveL 6524 to (-73.33, 55.91, -10) mm, rotated rx 180 ry 0 rz 90 deg; joints [74.994, -18.816, 90.444, 0, 18.372, 74.994]
  MoveL 6525 to (-73.33, 29.14, -10) mm, rotated rx 180 ry 0 rz 90 deg; joints [74.082, -18.708, 89.949, 0, 18.759, 74.082]
  MoveL 6526 to (-65.78, 29.14, -10) mm, rotated rx -180 ry 0 rz 90 deg; joints [74.154, -18.597, 89.443, 0, 19.153, 74.154]
  MoveL 6527 to (-65.78, 29.14, -7) mm, rotated rx 180 ry 0 rz 90 deg; joints [74.154, -18.754, 89.545, 0, 19.208, 74.154]
  Establecer velocidad (1000.0 mm/s)
  MoveL 6528 to (-65.78, 29.14, 10) mm, rotated rx 180 ry 0 rz 90 deg; joints [74.154, -19.642, 90.114, 0, 19.529, 74.154]
  Establecer velocidad (66.7 mm/s)
  MoveL 6529 to (-39.83, -32.22, 10) mm, rotated rx 180 ry 0 rz 90 deg; joints [72.375, -18.921, 87.095, 0, 21.827, 72.375]
  MoveL 6530 to (-39.83, -32.22, -6.75) mm, rotated rx -180 ry 0 rz 90 deg; joints [72.375, -18.058, 86.535, 0, 21.523, 72.375]
  MoveL 6531 to (-39.96, -30.71, -7.16) mm, rotated rx -180 ry 0 rz 90 deg; joints [72.423, -18.047, 86.563, 0, 21.484, 72.423]
  MoveL 6532 to (-40.45, -29.27, -7.56) mm, rotated rx 180 ry 0 rz 90 deg; joints [72.465, -18.042, 86.614, 0, 21.428, 72.465]
  MoveL 6533 to (-41.24, -27.98, -7.97) mm, rotated rx -180 ry 0 rz 90 deg; joints [72.499, -18.041, 86.683, 0, 21.358, 72.499]
  MoveL 6534 to (-42.3, -26.89, -8.37) mm, rotated rx 180 ry 0 rz 90 deg; joints [72.524, -18.043, 86.765, 0, 21.278, 72.524]
  MoveL 6535 to (-43.58, -26.06, -8.78) mm, rotated rx 180 ry 0 rz 90 deg; joints [72.538, -18.048, 86.857, 0, 21.191, 72.538]
  MoveL 6536 to (-45.01, -25.54, -9.19) mm, rotated rx 180 ry 0 rz 90 deg; joints [72.54, -18.053, 86.952, 0, 21.101, 72.54]
  MoveL 6537 to (-46.51, -25.34, -9.59) mm, rotated rx -180 ry 0 rz 90 deg; joints [72.531, -18.058, 87.045, 0, 21.013, 72.531]
  MoveL 6538 to (-48.02, -25.51, -10) mm, rotated rx 180 ry 0 rz 90 deg; joints [72.51, -18.061, 87.131, 0, 20.93, 72.51]
  MoveL 6539 to (-70.6, -30.23, -10) mm, rotated rx 180 ry 0 rz 90 deg; joints [72.117, -18.396, 88.558, 0, 19.838, 72.117]
